LIN {X 0,Y 417.232,Z 275.449,A -85,B 0,C 180,E1 -10353.741,E2 -10353.741} C_VEL
LIN {X 0,Y 417.731,Z 261.552,A -85,B 0,C 180,E1 -10354.25,E2 -10354.25} C_VEL
LIN {X 0,Y 418.018,Z 247.194,A -85,B 0,C 180,E1 -10354.579,E2 -10354.579} C_VEL
LIN {X 0,Y 419.623,Z 143.147,A -85,B 0,C 180,E1 -10356.374,E2 -10356.374} C_VEL
LIN {X 0,Y 414.972,Z 121.368,A -85,B 0,C 180,E1 -10357.003,E2 -10357.003} C_VEL
LIN {X 0,Y 414.069,Z 118.736,A -85,B 0,C 180,E1 -10357.128,E2 -10357.128} C_VEL
LIN {X 0,Y 411.674,Z 106.755,A -85,B 0,C 180,E1 -10359.828,E2 -10359.828} C_VEL
LIN {X 0,Y 411.268,Z 104.886,A -85,B 0,C 180,E1 -10360.273,E2 -10360.273} C_VEL
LIN {X 0,Y 411.343,Z 104.878,A -85,B 0,C 180,E1 -10363.149,E2 -10363.149} C_VEL
LIN {X 0,Y 411.264,Z 104.878,A -85,B 0,C 180,E1 -10366.887,E2 -10366.887} C_VEL
LIN {X 0,Y 411.218,Z 104.885,A -85,B 0,C 180,E1 -10369.986,E2 -10369.986} C_VEL
LIN {X 0,Y 411.195,Z 104.89,A -85,B 0,C 180,E1 -10373.146,E2 -10373.146} C_VEL
LIN {X 0,Y 411.203,Z 104.885,A -85,B 0,C 180,E1 -10376.382,E2 -10376.382} C_VEL
LIN {X 0,Y 411.177,Z 104.89,A -85,B 0,C 180,E1 -10379.713,E2 -10379.713} C_VEL
LIN {X 0,Y 411.172,Z 104.896,A -85,B 0,C 180,E1 -10383.157,E2 -10383.157} C_VEL
LIN {X 0,Y 411.199,Z 104.889,A -85,B 0,C 180,E1 -10386.739,E2 -10386.739} C_VEL
LIN {X 0,Y 411.205,Z 104.885,A -85,B 0,C 180,E1 -10389.734,E2 -10389.734} C_VEL
LIN {X 0,Y 411.197,Z 104.889,A -85,B 0,C 180,E1 -10393.128,E2 -10393.128} C_VEL
LIN {X 0,Y 411.218,Z 104.883,A -85,B 0,C 180,E1 -10395.872,E2 -10395.872} C_VEL
LIN {X 0,Y 411.184,Z 104.887,A -85,B 0,C 180,E1 -10399.502,E2 -10399.502} C_VEL
LIN {X 0,Y 411.178,Z 104.89,A -85,B 0,C 180,E1 -10402.03,E2 -10402.03} C_VEL
LIN {X 0,Y 411.179,Z 104.888,A -85,B 0,C 180,E1 -10405.669,E2 -10405.669} C_VEL
LIN {X 0,Y 411.176,Z 104.888,A -85,B 0,C 180,E1 -10409.156,E2 -10409.156} C_VEL
LIN {X 0,Y 411.236,Z 104.884,A -85,B 0,C 180,E1 -10412.525,E2 -10412.525} C_VEL
LIN {X 0,Y 411.21,Z 104.887,A -85,B 0,C 180,E1 -10415.788,E2 -10415.788} C_VEL
LIN {X 0,Y 411.224,Z 104.882,A -85,B 0,C 180,E1 -10418.972,E2 -10418.972} C_VEL
LIN {X 0,Y 411.235,Z 104.886,A -85,B 0,C 180,E1 -10422.088,E2 -10422.088} C_VEL
LIN {X 0,Y 411.249,Z 104.88,A -85,B 0,C 180,E1 -10425.151,E2 -10425.151} C_VEL
LIN {X 0,Y 411.284,Z 104.877,A -85,B 0,C 180,E1 -10428.171,E2 -10428.171} C_VEL
LIN {X 0,Y 411.467,Z 104.853,A -85,B 0,C 180,E1 -10432.15,E2 -10432.15} C_VEL
LIN {X 0,Y 411.465,Z 104.854,A -85,B 0,C 180,E1 -10434.121,E2 -10434.121} C_VEL
LIN {X 0,Y 411.503,Z 104.848,A -85,B 0,C 180,E1 -10438.046,E2 -10438.046} C_VEL
LIN {X 0,Y 411.633,Z 104.832,A -85,B 0,C 180,E1 -10440.003,E2 -10440.003} C_VEL
LIN {X 0,Y 411.457,Z 104.857,A -85,B 0,C 180,E1 -10442.94,E2 -10442.94} C_VEL
LIN {X 0,Y 411.452,Z 104.858,A -85,B 0,C 180,E1 -10446.87,E2 -10446.87} C_VEL
LIN {X 0,Y 411.286,Z 104.875,A -85,B 0,C 180,E1 -10449.842,E2 -10449.842} C_VEL
LIN {X 0,Y 411.298,Z 104.878,A -85,B 0,C 180,E1 -10453.107,E2 -10453.107} C_VEL
LIN {X 0,Y 411.252,Z 104.885,A -85,B 0,C 180,E1 -10456.892,E2 -10456.892} C_VEL
LIN {X 0,Y 411.226,Z 104.883,A -85,B 0,C 180,E1 -10459.99,E2 -10459.99} C_VEL
LIN {X 0,Y 411.199,Z 104.887,A -85,B 0,C 180,E1 -10463.15,E2 -10463.15} C_VEL
LIN {X 0,Y 411.235,Z 104.886,A -85,B 0,C 180,E1 -10466.384,E2 -10466.384} C_VEL
LIN {X 0,Y 411.198,Z 104.886,A -85,B 0,C 180,E1 -10469.715,E2 -10469.715} C_VEL
LIN {X 0,Y 411.205,Z 104.885,A -85,B 0,C 180,E1 -10473.158,E2 -10473.158} C_VEL
LIN {X 0,Y 411.192,Z 104.889,A -85,B 0,C 180,E1 -10476.555,E2 -10476.555} C_VEL
LIN {X 0,Y 411.212,Z 104.887,A -85,B 0,C 180,E1 -10479.73,E2 -10479.73} C_VEL
LIN {X 0,Y 411.173,Z 104.889,A -85,B 0,C 180,E1 -10483.136,E2 -10483.136} C_VEL
LIN {X 0,Y 411.168,Z 104.896,A -85,B 0,C 180,E1 -10485.884,E2 -10485.884} C_VEL
LIN {X 0,Y 411.164,Z 104.89,A -85,B 0,C 180,E1 -10488.774,E2 -10488.774} C_VEL
LIN {X 0,Y 411.191,Z 104.89,A -85,B 0,C 180,E1 -10492.028,E2 -10492.028} C_VEL
LIN {X 0,Y 411.208,Z 104.891,A -85,B 0,C 180,E1 -10495.669,E2 -10495.669} C_VEL
LIN {X 0,Y 411.193,Z 104.891,A -85,B 0,C 180,E1 -10499.155,E2 -10499.155} C_VEL
LIN {X 0,Y 411.272,Z 104.953,A -85,B 0,C 180,E1 -10500.26,E2 -10500.26} C_VEL
LIN {X 0,Y 414.489,Z 119.861,A -85,B 0,C 180,E1 -10503.302,E2 -10503.302} C_VEL
LIN {X 0,Y 415.269,Z 124.242,A -85,B 0,C 180,E1 -10504.166,E2 -10504.166} C_VEL
LIN {X 0,Y 414.279,Z 139.428,A -85,B 0,C 180,E1 -10506.93,E2 -10506.93} C_VEL
LIN {X 0,Y 419.416,Z 170.231,A -85,B 0,C 180,E1 -10507.745,E2 -10507.745} C_VEL
LIN {X 0,Y 417.748,Z 278.062,A -85,B 0,C 180,E1 -10509.634,E2 -10509.634} C_VEL
LIN {X 0,Y 417.18,Z 292.545,A -85,B 0,C 180,E1 -10510.087,E2 -10510.087} C_VEL
LIN {X 0,Y 416.418,Z 306.482,A -85,B 0,C 180,E1 -10510.723,E2 -10510.723} C_VEL
LIN {X 0,Y 415.61,Z 319.466,A -85,B 0,C 180,E1 -10511.516,E2 -10511.516} C_VEL
LIN {X 0,Y 414.604,Z 332.073,A -85,B 0,C 180,E1 -10512.491,E2 -10512.491} C_VEL
LIN {X 0,Y 413.679,Z 343.587,A -85,B 0,C 180,E1 -10513.596,E2 -10513.596} C_VEL
LIN {X 0,Y 412.83,Z 353.163,A -85,B 0,C 180,E1 -10514.702,E2 -10514.702} C_VEL
LIN {X 0,Y 412.028,Z 363.834,A -85,B 0,C 180,E1 -10516.186,E2 -10516.186} C_VEL
LIN {X 0,Y 411.333,Z 372.623,A -85,B 0,C 180,E1 -10517.67,E2 -10517.67} C_VEL
LIN {X 0,Y 410.717,Z 381.037,A -85,B 0,C 180,E1 -10519.402,E2 -10519.402} C_VEL
LIN {X 0,Y 410.328,Z 387.778,A -85,B 0,C 180,E1 -10521.134,E2 -10521.134} C_VEL
LIN {X 0,Y 410.063,Z 393.746,A -85,B 0,C 180,E1 -10523.111,E2 -10523.111} C_VEL
LIN {X 0,Y 409.972,Z 398.111,A -85,B 0,C 180,E1 -10525.084,E2 -10525.084} C_VEL
LIN {X 0,Y 409.917,Z 401.01,A -85,B 0,C 180,E1 -10527.053,E2 -10527.053} C_VEL
LIN {X 0,Y 409.937,Z 402.528,A -85,B 0,C 180,E1 -10529.019,E2 -10529.019} C_VEL
LIN {X 0,Y 409.937,Z 402.7,A -85,B 0,C 180,E1 -10530.984,E2 -10530.984} C_VEL
LIN {X 0,Y 409.913,Z 401.537,A -85,B 0,C 180,E1 -10532.95,E2 -10532.95} C_VEL
LIN {X 0,Y 409.982,Z 399.026,A -85,B 0,C 180,E1 -10534.918,E2 -10534.918} C_VEL
LIN {X 0,Y 410.092,Z 395.089,A -85,B 0,C 180,E1 -10536.891,E2 -10536.891} C_VEL
LIN {X 0,Y 410.402,Z 389.593,A -85,B 0,C 180,E1 -10538.867,E2 -10538.867} C_VEL
LIN {X 0,Y 410.803,Z 383.407,A -85,B 0,C 180,E1 -10540.599,E2 -10540.599} C_VEL
LIN {X 0,Y 411.606,Z 375.714,A -85,B 0,C 180,E1 -10542.325,E2 -10542.325} C_VEL
LIN {X 0,Y 412.283,Z 367.712,A -85,B 0,C 180,E1 -10543.808,E2 -10543.808} C_VEL
LIN {X 0,Y 413.236,Z 358.091,A -85,B 0,C 180,E1 -10545.286,E2 -10545.286} C_VEL
LIN {X 0,Y 414.334,Z 347.445,A -85,B 0,C 180,E1 -10546.634,E2 -10546.634} C_VEL
LIN {X 0,Y 415.594,Z 335.694,A -85,B 0,C 180,E1 -10547.85,E2 -10547.85} C_VEL
LIN {X 0,Y 416.616,Z 324.265,A -85,B 0,C 180,E1 -10548.819,E2 -10548.819} C_VEL
LIN {X 0,Y 417.625,Z 311.778,A -85,B 0,C 180,E1 -10549.669,E2 -10549.669} C_VEL
LIN {X 0,Y 418.607,Z 298.001,A -85,B 0,C 180,E1 -10550.389,E2 -10550.389} C_VEL
LIN {X 0,Y 419.4,Z 284.502,A -85,B 0,C 180,E1 -10550.894,E2 -10550.894} C_VEL
LIN {X 0,Y 419.898,Z 271.046,A -85,B 0,C 180,E1 -10551.221,E2 -10551.221} C_VEL
LIN {X 0,Y 421.535,Z 169.575,A -85,B 0,C 180,E1 -10553.015,E2 -10553.015} C_VEL
LIN {X 0,Y 417.055,Z 146.34,A -85,B 0,C 180,E1 -10553.757,E2 -10553.757} C_VEL
LIN {X 0,Y 415.437,Z 138.972,A -85,B 0,C 180,E1 -10554.021,E2 -10554.021} C_VEL
LIN {X 0,Y 416.422,Z 128.312,A -85,B 0,C 180,E1 -10556.029,E2 -10556.029} C_VEL
LIN {X 0,Y 414.54,Z 118.327,A -85,B 0,C 180,E1 -10558.162,E2 -10558.162} C_VEL
LIN {X 0,Y 411.687,Z 106.654,A -85,B 0,C 180,E1 -10560.808,E2 -10560.808} C_VEL
LIN {X 0,Y 411.202,Z 104.895,A -85,B 0,C 180,E1 -10561.238,E2 -10561.238} C_VEL
LIN {X 0,Y 411.205,Z 104.889,A -85,B 0,C 180,E1 -10564.335,E2 -10564.335} C_VEL
LIN {X 0,Y 411.202,Z 104.887,A -85,B 0,C 180,E1 -10566.742,E2 -10566.742} C_VEL
LIN {X 0,Y 411.209,Z 104.886,A -85,B 0,C 180,E1 -10569.724,E2 -10569.724} C_VEL
LIN {X 0,Y 411.185,Z 104.889,A -85,B 0,C 180,E1 -10573.134,E2 -10573.134} C_VEL
LIN {X 0,Y 411.182,Z 104.893,A -85,B 0,C 180,E1 -10575.881,E2 -10575.881} C_VEL
LIN {X 0,Y 411.174,Z 104.875,A -85,B 0,C 180,E1 -10578.772,E2 -10578.772} C_VEL
LIN {X 0,Y 411.2,Z 104.886,A -85,B 0,C 180,E1 -10582.024,E2 -10582.024} C_VEL
LIN {X 0,Y 411.217,Z 104.887,A -85,B 0,C 180,E1 -10585.122,E2 -10585.122} C_VEL
LIN {X 0,Y 411.179,Z 104.888,A -85,B 0,C 180,E1 -10588.001,E2 -10588.001} C_VEL
LIN {X 0,Y 411.207,Z 104.886,A -85,B 0,C 180,E1 -10591.407,E2 -10591.407} C_VEL
LIN {X 0,Y 411.241,Z 104.885,A -85,B 0,C 180,E1 -10594.928,E2 -10594.928} C_VEL
LIN {X 0,Y 411.218,Z 104.885,A -85,B 0,C 180,E1 -10597.912,E2 -10597.912} C_VEL
LIN {X 0,Y 411.232,Z 104.885,A -85,B 0,C 180,E1 -10601.049,E2 -10601.049} C_VEL
LIN {X 0,Y 411.266,Z 104.873,A -85,B 0,C 180,E1 -10604.129,E2 -10604.129} C_VEL
LIN {X 0,Y 411.315,Z 104.87,A -85,B 0,C 180,E1 -10607.163,E2 -10607.163} C_VEL
LIN {X 0,Y 411.301,Z 104.876,A -85,B 0,C 180,E1 -10610.159,E2 -10610.159} C_VEL
LIN {X 0,Y 411.402,Z 104.859,A -85,B 0,C 180,E1 -10613.129,E2 -10613.129} C_VEL
LIN {X 0,Y 411.308,Z 104.873,A -85,B 0,C 180,E1 -10615.096,E2 -10615.096} C_VEL
LIN {X 0,Y 411.516,Z 104.846,A -85,B 0,C 180,E1 -10618.039,E2 -10618.039} C_VEL
LIN {X 0,Y 411.643,Z 104.834,A -85,B 0,C 180,E1 -10619.997,E2 -10619.997} C_VEL
LIN {X 0,Y 411.456,Z 104.855,A -85,B 0,C 180,E1 -10622.934,E2 -10622.934} C_VEL
LIN {X 0,Y 411.428,Z 104.858,A -85,B 0,C 180,E1 -10626.864,E2 -10626.864} C_VEL
LIN {X 0,Y 411.294,Z 104.874,A -85,B 0,C 180,E1 -10629.835,E2 -10629.835} C_VEL
LIN {X 0,Y 411.307,Z 104.872,A -85,B 0,C 180,E1 -10633.1,E2 -10633.1} C_VEL
LIN {X 0,Y 411.257,Z 104.877,A -85,B 0,C 180,E1 -10636.885,E2 -10636.885} C_VEL
LIN {X 0,Y 411.228,Z 104.88,A -85,B 0,C 180,E1 -10639.983,E2 -10639.983} C_VEL
LIN {X 0,Y 411.191,Z 104.889,A -85,B 0,C 180,E1 -10643.144,E2 -10643.144} C_VEL
LIN {X 0,Y 411.227,Z 104.881,A -85,B 0,C 180,E1 -10646.377,E2 -10646.377} C_VEL
LIN {X 0,Y 411.192,Z 104.875,A -85,B 0,C 180,E1 -10649.709,E2 -10649.709} C_VEL
LIN {X 0,Y 411.196,Z 104.884,A -85,B 0,C 180,E1 -10653.152,E2 -10653.152} C_VEL
LIN {X 0,Y 411.179,Z 104.895,A -85,B 0,C 180,E1 -10656.548,E2 -10656.548} C_VEL
LIN {X 0,Y 411.194,Z 104.891,A -85,B 0,C 180,E1 -10659.723,E2 -10659.723} C_VEL
LIN {X 0,Y 411.156,Z 104.897,A -85,B 0,C 180,E1 -10663.13,E2 -10663.13} C_VEL
LIN {X 0,Y 411.16,Z 104.933,A -85,B 0,C 180,E1 -10666.378,E2 -10666.378} C_VEL
LIN {X 0,Y 413.745,Z 115.767,A -85,B 0,C 180,E1 -10669.096,E2 -10669.096} C_VEL
LIN {X 0,Y 414.472,Z 119.37,A -85,B 0,C 180,E1 -10669.967,E2 -10669.967} C_VEL
LIN {X 0,Y 418.585,Z 129.465,A -85,B 0,C 180,E1 -10670.453,E2 -10670.453} C_VEL
LIN {X 0,Y 422,Z 144.277,A -85,B 0,C 180,E1 -10670.966,E2 -10670.966} C_VEL
LIN {X 0,Y 419.998,Z 256.023,A -85,B 0,C 180,E1 -10672.956,E2 -10672.956} C_VEL
LIN {X 0,Y 419.376,Z 270.729,A -85,B 0,C 180,E1 -10673.419,E2 -10673.419} C_VEL
LIN {X 0,Y 418.604,Z 285.001,A -85,B 0,C 180,E1 -10674.085,E2 -10674.085} C_VEL
LIN {X 0,Y 417.765,Z 296.896,A -85,B 0,C 180,E1 -10674.816,E2 -10674.816} C_VEL
LIN {X 0,Y 416.802,Z 308.452,A -85,B 0,C 180,E1 -10675.704,E2 -10675.704} C_VEL
LIN {X 0,Y 415.673,Z 320.161,A -85,B 0,C 180,E1 -10676.811,E2 -10676.811} C_VEL
LIN {X 0,Y 414.582,Z 330.837,A -85,B 0,C 180,E1 -10678.042,E2 -10678.042} C_VEL
LIN {X 0,Y 413.566,Z 340.245,A -85,B 0,C 180,E1 -10679.347,E2 -10679.347} C_VEL
LIN {X 0,Y 412.538,Z 349.792,A -85,B 0,C 180,E1 -10680.952,E2 -10680.952} C_VEL
LIN {X 0,Y 411.715,Z 357.654,A -85,B 0,C 180,E1 -10682.568,E2 -10682.568} C_VEL
LIN {X 0,Y 411.116,Z 363.963,A -85,B 0,C 180,E1 -10684.155,E2 -10684.155} C_VEL
LIN {X 0,Y 410.655,Z 369.11,A -85,B 0,C 180,E1 -10685.747,E2 -10685.747} C_VEL
LIN {X 0,Y 410.33,Z 373.842,A -85,B 0,C 180,E1 -10687.639,E2 -10687.639} C_VEL
LIN {X 0,Y 410.094,Z 376.27,A -85,B 0,C 180,E1 -10688.905,E2 -10688.905} C_VEL
LIN {X 0,Y 409.88,Z 378.977,A -85,B 0,C 180,E1 -10690.986,E2 -10690.986} C_VEL
LIN {X 0,Y 409.79,Z 380.163,A -85,B 0,C 180,E1 -10693.048,E2 -10693.048} C_VEL
LIN {X 0,Y 409.814,Z 380.219,A -85,B 0,C 180,E1 -10694.073,E2 -10694.073} C_VEL
LIN {X 0,Y 409.789,Z 379.28,A -85,B 0,C 180,E1 -10696.106,E2 -10696.106} C_VEL
LIN {X 0,Y 409.959,Z 376.935,A -85,B 0,C 180,E1 -10698.127,E2 -10698.127} C_VEL
LIN {X 0,Y 410.151,Z 373.162,A -85,B 0,C 180,E1 -10700.132,E2 -10700.132} C_VEL
LIN {X 0,Y 410.382,Z 369.027,A -85,B 0,C 180,E1 -10701.722,E2 -10701.722} C_VEL
LIN {X 0,Y 409.855,Z 366.761,A -85,B 0,C 180,E1 -10702.481,E2 -10702.481} C_VEL
LIN {X 0,Y 407.293,Z 362.771,A -85,B 0,C 180,E1 -10703.703,E2 -10703.703} C_VEL
LIN {X 0,Y 404.787,Z 358.223,A -85,B 0,C 180,E1 -10704.898,E2 -10704.898} C_VEL
LIN {X 0,Y 404.353,Z 355.068,A -85,B 0,C 180,E1 -10705.605,E2 -10705.605} C_VEL
LIN {X 0,Y 405.15,Z 346.404,A -85,B 0,C 180,E1 -10707.264,E2 -10707.264} C_VEL
LIN {X 0,Y 406.01,Z 336.893,A -85,B 0,C 180,E1 -10708.759,E2 -10708.759} C_VEL
LIN {X 0,Y 406.95,Z 326.374,A -85,B 0,C 180,E1 -10710.122,E2 -10710.122} C_VEL
LIN {X 0,Y 407.826,Z 315.863,A -85,B 0,C 180,E1 -10711.251,E2 -10711.251} C_VEL
LIN {X 0,Y 408.785,Z 303.467,A -85,B 0,C 180,E1 -10712.339,E2 -10712.339} C_VEL
LIN {X 0,Y 409.661,Z 291.236,A -85,B 0,C 180,E1 -10713.195,E2 -10713.195} C_VEL
LIN {X 0,Y 410.372,Z 277.79,A -85,B 0,C 180,E1 -10713.927,E2 -10713.927} C_VEL
LIN {X 0,Y 410.892,Z 263.957,A -85,B 0,C 180,E1 -10714.474,E2 -10714.474} C_VEL
LIN {X 0,Y 411.246,Z 249.63,A -85,B 0,C 180,E1 -10714.839,E2 -10714.839} C_VEL
LIN {X 0,Y 412.995,Z 144.462,A -85,B 0,C 180,E1 -10716.679,E2 -10716.679} C_VEL
LIN {X 0,Y 408.494,Z 123.578,A -85,B 0,C 180,E1 -10717.293,E2 -10717.293} C_VEL
LIN {X 0,Y 406.945,Z 119.084,A -85,B 0,C 180,E1 -10717.459,E2 -10717.459} C_VEL
LIN {X 0,Y 404.703,Z 108.046,A -85,B 0,C 180,E1 -10719.999,E2 -10719.999} C_VEL
LIN {X 0,Y 404.227,Z 105.761,A -85,B 0,C 180,E1 -10720.58,E2 -10720.58} C_VEL
LIN {X 0,Y 404.284,Z 105.757,A -85,B 0,C 180,E1 -10723.244,E2 -10723.244} C_VEL
LIN {X 0,Y 404.211,Z 105.758,A -85,B 0,C 180,E1 -10727.191,E2 -10727.191} C_VEL
LIN {X 0,Y 404.17,Z 105.761,A -85,B 0,C 180,E1 -10730.35,E2 -10730.35} C_VEL
LIN {X 0,Y 404.149,Z 105.769,A -85,B 0,C 180,E1 -10733.574,E2 -10733.574} C_VEL
LIN {X 0,Y 404.16,Z 105.765,A -85,B 0,C 180,E1 -10736.878,E2 -10736.878} C_VEL
LIN {X 0,Y 404.121,Z 105.767,A -85,B 0,C 180,E1 -10740.285,E2 -10740.285} C_VEL
LIN {X 0,Y 404.112,Z 105.769,A -85,B 0,C 180,E1 -10743.813,E2 -10743.813} C_VEL
LIN {X 0,Y 404.145,Z 105.77,A -85,B 0,C 180,E1 -10746.885,E2 -10746.885} C_VEL
LIN {X 0,Y 404.165,Z 105.762,A -85,B 0,C 180,E1 -10750.09,E2 -10750.09} C_VEL
LIN {X 0,Y 404.171,Z 105.765,A -85,B 0,C 180,E1 -10753.093,E2 -10753.093} C_VEL
LIN {X 0,Y 404.19,Z 105.759,A -85,B 0,C 180,E1 -10755.938,E2 -10755.938} C_VEL
LIN {X 0,Y 404.137,Z 105.772,A -85,B 0,C 180,E1 -10758.643,E2 -10758.643} C_VEL
LIN {X 0,Y 404.135,Z 105.765,A -85,B 0,C 180,E1 -10761.493,E2 -10761.493} C_VEL
LIN {X 0,Y 404.158,Z 105.764,A -85,B 0,C 180,E1 -10764.987,E2 -10764.987} C_VEL
LIN {X 0,Y 404.125,Z 105.771,A -85,B 0,C 180,E1 -10768.557,E2 -10768.557} C_VEL
LIN {X 0,Y 404.174,Z 105.765,A -85,B 0,C 180,E1 -10772.004,E2 -10772.004} C_VEL
LIN {X 0,Y 404.158,Z 105.763,A -85,B 0,C 180,E1 -10775.338,E2 -10775.338} C_VEL
LIN {X 0,Y 404.182,Z 105.761,A -85,B 0,C 180,E1 -10778.587,E2 -10778.587} C_VEL
LIN {X 0,Y 404.197,Z 105.763,A -85,B 0,C 180,E1 -10781.765,E2 -10781.765} C_VEL
LIN {X 0,Y 404.195,Z 105.758,A -85,B 0,C 180,E1 -10784.886,E2 -10784.886} C_VEL
LIN {X 0,Y 404.254,Z 105.755,A -85,B 0,C 180,E1 -10787.962,E2 -10787.962} C_VEL
LIN {X 0,Y 404.419,Z 105.732,A -85,B 0,C 180,E1 -10792.103,E2 -10792.103} C_VEL
LIN {X 0,Y 404.413,Z 105.733,A -85,B 0,C 180,E1 -10794.018,E2 -10794.018} C_VEL
LIN {X 0,Y 404.472,Z 105.725,A -85,B 0,C 180,E1 -10798.012,E2 -10798.012} C_VEL
LIN {X 0,Y 404.602,Z 105.708,A -85,B 0,C 180,E1 -10800.003,E2 -10800.003} C_VEL
LIN {X 0,Y 404.414,Z 105.734,A -85,B 0,C 180,E1 -10802.992,E2 -10802.992} C_VEL
LIN {X 0,Y 404.403,Z 105.737,A -85,B 0,C 180,E1 -10806.99,E2 -10806.99} C_VEL
LIN {X 0,Y 404.251,Z 105.751,A -85,B 0,C 180,E1 -10810.015,E2 -10810.015} C_VEL
LIN {X 0,Y 404.26,Z 105.754,A -85,B 0,C 180,E1 -10813.214,E2 -10813.214} C_VEL
LIN {X 0,Y 404.21,Z 105.761,A -85,B 0,C 180,E1 -10817.01,E2 -10817.01} C_VEL
LIN {X 0,Y 404.159,Z 105.765,A -85,B 0,C 180,E1 -10820.355,E2 -10820.355} C_VEL
LIN {X 0,Y 404.166,Z 105.762,A -85,B 0,C 180,E1 -10823.577,E2 -10823.577} C_VEL
LIN {X 0,Y 404.181,Z 105.76,A -85,B 0,C 180,E1 -10825.769,E2 -10825.769} C_VEL
LIN {X 0,Y 404.193,Z 105.76,A -85,B 0,C 180,E1 -10828.002,E2 -10828.002} C_VEL
LIN {X 0,Y 404.137,Z 105.765,A -85,B 0,C 180,E1 -10831.561,E2 -10831.561} C_VEL
LIN {X 0,Y 404.184,Z 105.76,A -85,B 0,C 180,E1 -10835.019,E2 -10835.019} C_VEL
LIN {X 0,Y 404.153,Z 105.764,A -85,B 0,C 180,E1 -10838.76,E2 -10838.76} C_VEL
LIN {X 0,Y 404.122,Z 105.769,A -85,B 0,C 180,E1 -10841.602,E2 -10841.602} C_VEL
LIN {X 0,Y 404.146,Z 105.765,A -85,B 0,C 180,E1 -10844.524,E2 -10844.524} C_VEL
LIN {X 0,Y 404.137,Z 105.766,A -85,B 0,C 180,E1 -10847.298,E2 -10847.298} C_VEL
LIN {X 0,Y 404.171,Z 105.766,A -85,B 0,C 180,E1 -10849.958,E2 -10849.958} C_VEL
LIN {X 0,Y 404.137,Z 105.766,A -85,B 0,C 180,E1 -10853.128,E2 -10853.128} C_VEL
LIN {X 0,Y 404.148,Z 105.769,A -85,B 0,C 180,E1 -10856.19,E2 -10856.19} C_VEL
LIN {X 0,Y 404.216,Z 105.941,A -85,B 0,C 180,E1 -10859.994,E2 -10859.994} C_VEL
LIN {X 0,Y 407.453,Z 120.771,A -85,B 0,C 180,E1 -10863.08,E2 -10863.08} C_VEL
LIN {X 0,Y 408.357,Z 126.76,A -85,B 0,C 180,E1 -10864.273,E2 -10864.273} C_VEL
LIN {X 0,Y 407.418,Z 139.188,A -85,B 0,C 180,E1 -10866.567,E2 -10866.567} C_VEL
LIN {X 0,Y 412.694,Z 170.64,A -85,B 0,C 180,E1 -10867.427,E2 -10867.427} C_VEL
LIN {X 0,Y 411.015,Z 277.225,A -85,B 0,C 180,E1 -10869.318,E2 -10869.318} C_VEL
LIN {X 0,Y 410.441,Z 291.926,A -85,B 0,C 180,E1 -10869.779,E2 -10869.779} C_VEL
LIN {X 0,Y 409.66,Z 305.399,A -85,B 0,C 180,E1 -10870.393,E2 -10870.393} C_VEL
LIN {X 0,Y 408.764,Z 318.886,A -85,B 0,C 180,E1 -10871.218,E2 -10871.218} C_VEL
LIN {X 0,Y 407.786,Z 331.318,A -85,B 0,C 180,E1 -10872.189,E2 -10872.189} C_VEL
LIN {X 0,Y 406.78,Z 342.927,A -85,B 0,C 180,E1 -10873.309,E2 -10873.309} C_VEL
LIN {X 0,Y 405.899,Z 352.583,A -85,B 0,C 180,E1 -10874.434,E2 -10874.434} C_VEL
LIN {X 0,Y 405.053,Z 363.318,A -85,B 0,C 180,E1 -10875.943,E2 -10875.943} C_VEL
LIN {X 0,Y 404.36,Z 372.163,A -85,B 0,C 180,E1 -10877.454,E2 -10877.454} C_VEL
LIN {X 0,Y 403.677,Z 380.63,A -85,B 0,C 180,E1 -10879.215,E2 -10879.215} C_VEL
LIN {X 0,Y 403.277,Z 387.426,A -85,B 0,C 180,E1 -10880.978,E2 -10880.978} C_VEL
LIN {X 0,Y 403.041,Z 392.086,A -85,B 0,C 180,E1 -10882.487,E2 -10882.487} C_VEL
LIN {X 0,Y 402.858,Z 396.38,A -85,B 0,C 180,E1 -10884.252,E2 -10884.252} C_VEL
LIN {X 0,Y 402.827,Z 399.477,A -85,B 0,C 180,E1 -10886,E2 -10886} C_VEL
LIN {X 0,Y 402.864,Z 401.709,A -85,B 0,C 180,E1 -10888.002,E2 -10888.002} C_VEL
LIN {X 0,Y 402.855,Z 402.579,A -85,B 0,C 180,E1 -10890.001,E2 -10890.001} C_VEL
LIN {X 0,Y 402.864,Z 402.111,A -85,B 0,C 180,E1 -10892.001,E2 -10892.001} C_VEL
LIN {X 0,Y 402.828,Z 400.306,A -85,B 0,C 180,E1 -10894.003,E2 -10894.003} C_VEL
LIN {X 0,Y 402.927,Z 397.133,A -85,B 0,C 180,E1 -10896.009,E2 -10896.009} C_VEL
LIN {X 0,Y 403.158,Z 392.478,A -85,B 0,C 180,E1 -10898.018,E2 -10898.018} C_VEL
LIN {X 0,Y 403.607,Z 386.192,A -85,B 0,C 180,E1 -10900.029,E2 -10900.029} C_VEL
LIN {X 0,Y 404.266,Z 379.215,A -85,B 0,C 180,E1 -10901.788,E2 -10901.788} C_VEL
LIN {X 0,Y 405.032,Z 370.917,A -85,B 0,C 180,E1 -10903.487,E2 -10903.487} C_VEL
LIN {X 0,Y 405.998,Z 361.607,A -85,B 0,C 180,E1 -10905.051,E2 -10905.051} C_VEL
LIN {X 0,Y 407.193,Z 350.766,A -85,B 0,C 180,E1 -10906.547,E2 -10906.547} C_VEL
LIN {X 0,Y 408.421,Z 339.795,A -85,B 0,C 180,E1 -10907.786,E2 -10907.786} C_VEL
LIN {X 0,Y 409.635,Z 327.789,A -85,B 0,C 180,E1 -10908.896,E2 -10908.896} C_VEL
LIN {X 0,Y 410.805,Z 314.957,A -85,B 0,C 180,E1 -10909.842,E2 -10909.842} C_VEL
LIN {X 0,Y 411.858,Z 301.474,A -85,B 0,C 180,E1 -10910.608,E2 -10910.608} C_VEL
LIN {X 0,Y 412.702,Z 287.662,A -85,B 0,C 180,E1 -10911.184,E2 -10911.184} C_VEL
LIN {X 0,Y 413.377,Z 273.369,A -85,B 0,C 180,E1 -10911.572,E2 -10911.572} C_VEL
LIN {X 0,Y 415.22,Z 170.983,A -85,B 0,C 180,E1 -10913.412,E2 -10913.412} C_VEL
LIN {X 0,Y 410.929,Z 148.637,A -85,B 0,C 180,E1 -10914.145,E2 -10914.145} C_VEL
LIN {X 0,Y 408.768,Z 138.757,A -85,B 0,C 180,E1 -10914.506,E2 -10914.506} C_VEL
LIN {X 0,Y 409.619,Z 129.836,A -85,B 0,C 180,E1 -10916.22,E2 -10916.22} C_VEL
LIN {X 0,Y 407.649,Z 119.651,A -85,B 0,C 180,E1 -10918.444,E2 -10918.444} C_VEL
LIN {X 0,Y 404.757,Z 108.233,A -85,B 0,C 180,E1 -10921.103,E2 -10921.103} C_VEL
LIN {X 0,Y 404.15,Z 105.772,A -85,B 0,C 180,E1 -10921.716,E2 -10921.716} C_VEL
LIN {X 0,Y 404.187,Z 105.762,A -85,B 0,C 180,E1 -10925.017,E2 -10925.017} C_VEL
LIN {X 0,Y 404.156,Z 105.768,A -85,B 0,C 180,E1 -10928.758,E2 -10928.758} C_VEL
LIN {X 0,Y 404.131,Z 105.767,A -85,B 0,C 180,E1 -10931.598,E2 -10931.598} C_VEL
LIN {X 0,Y 404.159,Z 105.766,A -85,B 0,C 180,E1 -10934.521,E2 -10934.521} C_VEL
LIN {X 0,Y 404.149,Z 105.766,A -85,B 0,C 180,E1 -10937.295,E2 -10937.295} C_VEL
LIN {X 0,Y 404.147,Z 105.76,A -85,B 0,C 180,E1 -10939.95,E2 -10939.95} C_VEL
LIN {X 0,Y 404.148,Z 105.763,A -85,B 0,C 180,E1 -10943.125,E2 -10943.125} C_VEL
LIN {X 0,Y 404.152,Z 105.764,A -85,B 0,C 180,E1 -10946.186,E2 -10946.186} C_VEL
LIN {X 0,Y 404.158,Z 105.767,A -85,B 0,C 180,E1 -10949.713,E2 -10949.713} C_VEL
LIN {X 0,Y 404.149,Z 105.765,A -85,B 0,C 180,E1 -10953.117,E2 -10953.117} C_VEL
LIN {X 0,Y 404.174,Z 105.756,A -85,B 0,C 180,E1 -10956.423,E2 -10956.423} C_VEL
LIN {X 0,Y 404.205,Z 105.751,A -85,B 0,C 180,E1 -10959.872,E2 -10959.872} C_VEL
LIN {X 0,Y 404.229,Z 105.754,A -85,B 0,C 180,E1 -10962.991,E2 -10962.991} C_VEL
LIN {X 0,Y 404.295,Z 105.747,A -85,B 0,C 180,E1 -10966.936,E2 -10966.936} C_VEL
LIN {X 0,Y 404.267,Z 105.751,A -85,B 0,C 180,E1 -10969.986,E2 -10969.986} C_VEL
LIN {X 0,Y 404.353,Z 105.738,A -85,B 0,C 180,E1 -10973.009,E2 -10973.009} C_VEL
LIN {X 0,Y 404.279,Z 105.749,A -85,B 0,C 180,E1 -10975.01,E2 -10975.01} C_VEL
LIN {X 0,Y 404.485,Z 105.722,A -85,B 0,C 180,E1 -10978.005,E2 -10978.005} C_VEL
LIN {X 0,Y 404.613,Z 105.709,A -85,B 0,C 180,E1 -10979.997,E2 -10979.997} C_VEL
LIN {X 0,Y 404.414,Z 105.732,A -85,B 0,C 180,E1 -10982.985,E2 -10982.985} C_VEL
LIN {X 0,Y 404.374,Z 105.737,A -85,B 0,C 180,E1 -10986.984,E2 -10986.984} C_VEL
LIN {X 0,Y 404.26,Z 105.751,A -85,B 0,C 180,E1 -10990.008,E2 -10990.008} C_VEL
LIN {X 0,Y 404.268,Z 105.748,A -85,B 0,C 180,E1 -10993.207,E2 -10993.207} C_VEL
LIN {X 0,Y 404.216,Z 105.754,A -85,B 0,C 180,E1 -10997.003,E2 -10997.003} C_VEL
LIN {X 0,Y 404.161,Z 105.76,A -85,B 0,C 180,E1 -11000.347,E2 -11000.347} C_VEL
LIN {X 0,Y 404.155,Z 105.766,A -85,B 0,C 180,E1 -11003.571,E2 -11003.571} C_VEL
LIN {X 0,Y 404.175,Z 105.759,A -85,B 0,C 180,E1 -11005.762,E2 -11005.762} C_VEL
LIN {X 0,Y 404.188,Z 105.76,A -85,B 0,C 180,E1 -11007.995,E2 -11007.995} C_VEL
LIN {X 0,Y 404.13,Z 105.77,A -85,B 0,C 180,E1 -11011.554,E2 -11011.554} C_VEL
LIN {X 0,Y 404.171,Z 105.759,A -85,B 0,C 180,E1 -11015.012,E2 -11015.012} C_VEL
LIN {X 0,Y 404.136,Z 105.767,A -85,B 0,C 180,E1 -11018.753,E2 -11018.753} C_VEL
LIN {X 0,Y 404.106,Z 105.771,A -85,B 0,C 180,E1 -11021.595,E2 -11021.595} C_VEL
LIN {X 0,Y 404.127,Z 105.775,A -85,B 0,C 180,E1 -11024.518,E2 -11024.518} C_VEL
LIN {X 0,Y 404.145,Z 105.938,A -85,B 0,C 180,E1 -11025.966,E2 -11025.966} C_VEL
LIN {X 0,Y 406.975,Z 117.731,A -85,B 0,C 180,E1 -11028.986,E2 -11028.986} C_VEL
LIN {X 0,Y 407.353,Z 119.607,A -85,B 0,C 180,E1 -11029.447,E2 -11029.447} C_VEL
LIN {X 0,Y 412.681,Z 132.468,A -85,B 0,C 180,E1 -11030.092,E2 -11030.092} C_VEL
LIN {X 0,Y 415.605,Z 145.213,A -85,B 0,C 180,E1 -11030.547,E2 -11030.547} C_VEL
LIN {X 0,Y 413.545,Z 256.542,A -85,B 0,C 180,E1 -11032.565,E2 -11032.565} C_VEL
LIN {X 0,Y 412.881,Z 271.072,A -85,B 0,C 180,E1 -11033.03,E2 -11033.03} C_VEL
LIN {X 0,Y 412.037,Z 285.662,A -85,B 0,C 180,E1 -11033.724,E2 -11033.724} C_VEL
LIN {X 0,Y 410.996,Z 299.19,A -85,B 0,C 180,E1 -11034.587,E2 -11034.587} C_VEL
LIN {X 0,Y 409.814,Z 312.493,A -85,B 0,C 180,E1 -11035.681,E2 -11035.681} C_VEL
LIN {X 0,Y 408.558,Z 324.253,A -85,B 0,C 180,E1 -11036.891,E2 -11036.891} C_VEL
LIN {X 0,Y 407.368,Z 335.027,A -85,B 0,C 180,E1 -11038.25,E2 -11038.25} C_VEL
LIN {X 0,Y 406.395,Z 343.983,A -85,B 0,C 180,E1 -11039.612,E2 -11039.612} C_VEL
LIN {X 0,Y 405.331,Z 352.854,A -85,B 0,C 180,E1 -11041.238,E2 -11041.238} C_VEL
LIN {X 0,Y 404.628,Z 359.542,A -85,B 0,C 180,E1 -11042.718,E2 -11042.718} C_VEL
LIN {X 0,Y 404.024,Z 365.185,A -85,B 0,C 180,E1 -11044.221,E2 -11044.221} C_VEL
LIN {X 0,Y 403.564,Z 370.112,A -85,B 0,C 180,E1 -11045.841,E2 -11045.841} C_VEL
LIN {X 0,Y 403.269,Z 373.989,A -85,B 0,C 180,E1 -11047.454,E2 -11047.454} C_VEL
LIN {X 0,Y 402.917,Z 377.674,A -85,B 0,C 180,E1 -11049.581,E2 -11049.581} C_VEL
LIN {X 0,Y 402.851,Z 378.928,A -85,B 0,C 180,E1 -11050.641,E2 -11050.641} C_VEL
LIN {X 0,Y 402.684,Z 380.318,A -85,B 0,C 180,E1 -11052.739,E2 -11052.739} C_VEL
LIN {X 0,Y 402.697,Z 380.237,A -85,B 0,C 180,E1 -11054.823,E2 -11054.823} C_VEL
LIN {X 0,Y 402.718,Z 378.75,A -85,B 0,C 180,E1 -11056.886,E2 -11056.886} C_VEL
LIN {X 0,Y 402.95,Z 375.846,A -85,B 0,C 180,E1 -11058.938,E2 -11058.938} C_VEL
LIN {X 0,Y 403.179,Z 371.486,A -85,B 0,C 180,E1 -11060.973,E2 -11060.973} C_VEL
LIN {X 0,Y 403.609,Z 365.538,A -85,B 0,C 180,E1 -11062.997,E2 -11062.997} C_VEL
LIN {X 0,Y 404.049,Z 358.858,A -85,B 0,C 180,E1 -11064.759,E2 -11064.759} C_VEL
LIN {X 0,Y 404.353,Z 355.068,A -85,B 0,C 180,E1 -11065.605,E2 -11065.605} C_VEL
LIN {X 0,Y 403.952,Z 351.786,A -85,B 0,C 180,E1 -11066.296,E2 -11066.296} C_VEL
LIN {X 0,Y 401.644,Z 346.163,A -85,B 0,C 180,E1 -11067.415,E2 -11067.415} C_VEL
LIN {X 0,Y 399.424,Z 340.131,A -85,B 0,C 180,E1 -11068.494,E2 -11068.494} C_VEL
LIN {X 0,Y 399.159,Z 336.081,A -85,B 0,C 180,E1 -11069.112,E2 -11069.112} C_VEL
LIN {X 0,Y 400.153,Z 325.322,A -85,B 0,C 180,E1 -11070.502,E2 -11070.502} C_VEL
LIN {X 0,Y 401.147,Z 313.273,A -85,B 0,C 180,E1 -11071.774,E2 -11071.774} C_VEL
LIN {X 0,Y 402.14,Z 301.773,A -85,B 0,C 180,E1 -11072.753,E2 -11072.753} C_VEL
LIN {X 0,Y 403.033,Z 288.089,A -85,B 0,C 180,E1 -11073.685,E2 -11073.685} C_VEL
LIN {X 0,Y 403.723,Z 274.101,A -85,B 0,C 180,E1 -11074.398,E2 -11074.398} C_VEL
LIN {X 0,Y 404.246,Z 260.338,A -85,B 0,C 180,E1 -11074.892,E2 -11074.892} C_VEL
LIN {X 0,Y 404.624,Z 243.267,A -85,B 0,C 180,E1 -11075.262,E2 -11075.262} C_VEL
LIN {X 0,Y 406.239,Z 145.253,A -85,B 0,C 180,E1 -11077.006,E2 -11077.006} C_VEL
LIN {X 0,Y 402.23,Z 126.279,A -85,B 0,C 180,E1 -11077.572,E2 -11077.572} C_VEL
LIN {X 0,Y 399.782,Z 119.188,A -85,B 0,C 180,E1 -11077.861,E2 -11077.861} C_VEL
LIN {X 0,Y 397.204,Z 106.636,A -85,B 0,C 180,E1 -11080.834,E2 -11080.834} C_VEL
LIN {X 0,Y 397.234,Z 106.634,A -85,B 0,C 180,E1 -11083.348,E2 -11083.348} C_VEL
LIN {X 0,Y 397.19,Z 106.633,A -85,B 0,C 180,E1 -11087.176,E2 -11087.176} C_VEL
LIN {X 0,Y 397.121,Z 106.639,A -85,B 0,C 180,E1 -11090.727,E2 -11090.727} C_VEL
LIN {X 0,Y 397.105,Z 106.642,A -85,B 0,C 180,E1 -11094.018,E2 -11094.018} C_VEL
LIN {X 0,Y 397.159,Z 106.64,A -85,B 0,C 180,E1 -11097.391,E2 -11097.391} C_VEL
LIN {X 0,Y 397.054,Z 106.651,A -85,B 0,C 180,E1 -11100.883,E2 -11100.883} C_VEL
LIN {X 0,Y 397.095,Z 106.644,A -85,B 0,C 180,E1 -11104.494,E2 -11104.494} C_VEL
LIN {X 0,Y 397.118,Z 106.64,A -85,B 0,C 180,E1 -11108.271,E2 -11108.271} C_VEL
LIN {X 0,Y 397.125,Z 106.639,A -85,B 0,C 180,E1 -11111.996,E2 -11111.996} C_VEL
LIN {X 0,Y 397.147,Z 106.639,A -85,B 0,C 180,E1 -11115.058,E2 -11115.058} C_VEL
LIN {X 0,Y 397.128,Z 106.639,A -85,B 0,C 180,E1 -11118.009,E2 -11118.009} C_VEL
LIN {X 0,Y 397.082,Z 106.644,A -85,B 0,C 180,E1 -11121.729,E2 -11121.729} C_VEL
LIN {X 0,Y 397.099,Z 106.642,A -85,B 0,C 180,E1 -11125.51,E2 -11125.51} C_VEL
LIN {X 0,Y 397.066,Z 106.646,A -85,B 0,C 180,E1 -11129.122,E2 -11129.122} C_VEL
LIN {X 0,Y 397.172,Z 106.635,A -85,B 0,C 180,E1 -11132.613,E2 -11132.613} C_VEL
LIN {X 0,Y 397.12,Z 106.645,A -85,B 0,C 180,E1 -11135.985,E2 -11135.985} C_VEL
LIN {X 0,Y 397.138,Z 106.638,A -85,B 0,C 180,E1 -11139.276,E2 -11139.276} C_VEL
LIN {X 0,Y 397.165,Z 106.634,A -85,B 0,C 180,E1 -11142.847,E2 -11142.847} C_VEL
LIN {X 0,Y 397.166,Z 106.639,A -85,B 0,C 180,E1 -11145.66,E2 -11145.66} C_VEL
LIN {X 0,Y 397.195,Z 106.63,A -85,B 0,C 180,E1 -11148.78,E2 -11148.78} C_VEL
LIN {X 0,Y 397.38,Z 106.609,A -85,B 0,C 180,E1 -11152.044,E2 -11152.044} C_VEL
LIN {X 0,Y 397.246,Z 106.625,A -85,B 0,C 180,E1 -11154.929,E2 -11154.929} C_VEL
LIN {X 0,Y 397.441,Z 106.601,A -85,B 0,C 180,E1 -11157.977,E2 -11157.977} C_VEL
LIN {X 0,Y 397.572,Z 106.584,A -85,B 0,C 180,E1 -11160.003,E2 -11160.003} C_VEL
LIN {X 0,Y 397.373,Z 106.612,A -85,B 0,C 180,E1 -11163.045,E2 -11163.045} C_VEL
LIN {X 0,Y 397.356,Z 106.617,A -85,B 0,C 180,E1 -11167.115,E2 -11167.115} C_VEL
LIN {X 0,Y 397.211,Z 106.628,A -85,B 0,C 180,E1 -11170.194,E2 -11170.194} C_VEL
LIN {X 0,Y 397.22,Z 106.629,A -85,B 0,C 180,E1 -11173.324,E2 -11173.324} C_VEL
LIN {X 0,Y 397.176,Z 106.635,A -85,B 0,C 180,E1 -11177.158,E2 -11177.158} C_VEL
LIN {X 0,Y 397.098,Z 106.649,A -85,B 0,C 180,E1 -11180.733,E2 -11180.733} C_VEL
LIN {X 0,Y 397.13,Z 106.639,A -85,B 0,C 180,E1 -11184.021,E2 -11184.021} C_VEL
LIN {X 0,Y 397.192,Z 106.63,A -85,B 0,C 180,E1 -11187.393,E2 -11187.393} C_VEL
LIN {X 0,Y 397.076,Z 106.647,A -85,B 0,C 180,E1 -11190.885,E2 -11190.885} C_VEL
LIN {X 0,Y 397.124,Z 106.643,A -85,B 0,C 180,E1 -11194.496,E2 -11194.496} C_VEL
LIN {X 0,Y 397.102,Z 106.647,A -85,B 0,C 180,E1 -11198.278,E2 -11198.278} C_VEL
LIN {X 0,Y 397.088,Z 106.643,A -85,B 0,C 180,E1 -11200.911,E2 -11200.911} C_VEL
LIN {X 0,Y 397.101,Z 106.645,A -85,B 0,C 180,E1 -11203.651,E2 -11203.651} C_VEL
LIN {X 0,Y 397.103,Z 106.642,A -85,B 0,C 180,E1 -11206.524,E2 -11206.524} C_VEL
LIN {X 0,Y 397.114,Z 106.641,A -85,B 0,C 180,E1 -11210.425,E2 -11210.425} C_VEL
LIN {X 0,Y 397.11,Z 106.642,A -85,B 0,C 180,E1 -11214.268,E2 -11214.268} C_VEL
LIN {X 0,Y 397.117,Z 106.642,A -85,B 0,C 180,E1 -11216.729,E2 -11216.729} C_VEL
LIN {X 0,Y 397.148,Z 106.773,A -85,B 0,C 180,E1 -11219.688,E2 -11219.688} C_VEL
LIN {X 0,Y 400.125,Z 120.203,A -85,B 0,C 180,E1 -11222.546,E2 -11222.546} C_VEL
LIN {X 0,Y 401.43,Z 127.533,A -85,B 0,C 180,E1 -11224.046,E2 -11224.046} C_VEL
LIN {X 0,Y 400.563,Z 138.989,A -85,B 0,C 180,E1 -11226.202,E2 -11226.202} C_VEL
LIN {X 0,Y 405.996,Z 171.872,A -85,B 0,C 180,E1 -11227.117,E2 -11227.117} C_VEL
LIN {X 0,Y 404.262,Z 277.392,A -85,B 0,C 180,E1 -11229.023,E2 -11229.023} C_VEL
LIN {X 0,Y 403.644,Z 291.976,A -85,B 0,C 180,E1 -11229.49,E2 -11229.49} C_VEL
LIN {X 0,Y 402.829,Z 305.386,A -85,B 0,C 180,E1 -11230.112,E2 -11230.112} C_VEL
LIN {X 0,Y 401.906,Z 319.106,A -85,B 0,C 180,E1 -11230.97,E2 -11230.97} C_VEL
LIN {X 0,Y 400.844,Z 331.987,A -85,B 0,C 180,E1 -11232.002,E2 -11232.002} C_VEL
LIN {X 0,Y 399.811,Z 343.455,A -85,B 0,C 180,E1 -11233.141,E2 -11233.141} C_VEL
LIN {X 0,Y 398.832,Z 353.978,A -85,B 0,C 180,E1 -11234.413,E2 -11234.413} C_VEL
LIN {X 0,Y 397.979,Z 364.318,A -85,B 0,C 180,E1 -11235.928,E2 -11235.928} C_VEL
LIN {X 0,Y 397.237,Z 373.063,A -85,B 0,C 180,E1 -11237.485,E2 -11237.485} C_VEL
LIN {X 0,Y 396.558,Z 381.28,A -85,B 0,C 180,E1 -11239.277,E2 -11239.277} C_VEL
LIN {X 0,Y 396.216,Z 387.062,A -85,B 0,C 180,E1 -11240.816,E2 -11240.816} C_VEL
LIN {X 0,Y 395.969,Z 391.753,A -85,B 0,C 180,E1 -11242.352,E2 -11242.352} C_VEL
LIN {X 0,Y 395.791,Z 395.637,A -85,B 0,C 180,E1 -11243.937,E2 -11243.937} C_VEL
LIN {X 0,Y 395.749,Z 399.212,A -85,B 0,C 180,E1 -11245.928,E2 -11245.928} C_VEL
LIN {X 0,Y 395.763,Z 401.475,A -85,B 0,C 180,E1 -11247.966,E2 -11247.966} C_VEL
LIN {X 0,Y 395.782,Z 402.376,A -85,B 0,C 180,E1 -11250.001,E2 -11250.001} C_VEL
LIN {X 0,Y 395.761,Z 401.937,A -85,B 0,C 180,E1 -11252.037,E2 -11252.037} C_VEL
LIN {X 0,Y 395.751,Z 400.162,A -85,B 0,C 180,E1 -11254.075,E2 -11254.075} C_VEL
LIN {X 0,Y 395.869,Z 396.928,A -85,B 0,C 180,E1 -11256.168,E2 -11256.168} C_VEL
LIN {X 0,Y 396.092,Z 392.41,A -85,B 0,C 180,E1 -11258.162,E2 -11258.162} C_VEL
LIN {X 0,Y 396.572,Z 386.162,A -85,B 0,C 180,E1 -11260.209,E2 -11260.209} C_VEL
LIN {X 0,Y 397.265,Z 379.235,A -85,B 0,C 180,E1 -11261.999,E2 -11261.999} C_VEL
LIN {X 0,Y 398.045,Z 371.506,A -85,B 0,C 180,E1 -11263.631,E2 -11263.631} C_VEL
LIN {X 0,Y 399.109,Z 361.755,A -85,B 0,C 180,E1 -11265.317,E2 -11265.317} C_VEL
LIN {X 0,Y 400.131,Z 352.929,A -85,B 0,C 180,E1 -11266.585,E2 -11266.585} C_VEL
LIN {X 0,Y 401.548,Z 341.263,A -85,B 0,C 180,E1 -11267.969,E2 -11267.969} C_VEL
LIN {X 0,Y 402.793,Z 329.616,A -85,B 0,C 180,E1 -11269.097,E2 -11269.097} C_VEL
LIN {X 0,Y 404.018,Z 317.355,A -85,B 0,C 180,E1 -11270.054,E2 -11270.054} C_VEL
LIN {X 0,Y 405.08,Z 304.654,A -85,B 0,C 180,E1 -11270.836,E2 -11270.836} C_VEL
LIN {X 0,Y 406.057,Z 290.622,A -85,B 0,C 180,E1 -11271.481,E2 -11271.481} C_VEL
LIN {X 0,Y 406.849,Z 275.7,A -85,B 0,C 180,E1 -11271.936,E2 -11271.936} C_VEL
LIN {X 0,Y 408.781,Z 171.391,A -85,B 0,C 180,E1 -11273.854,E2 -11273.854} C_VEL
LIN {X 0,Y 404.465,Z 149.255,A -85,B 0,C 180,E1 -11274.607,E2 -11274.607} C_VEL
LIN {X 0,Y 402.101,Z 138.487,A -85,B 0,C 180,E1 -11275.024,E2 -11275.024} C_VEL
LIN {X 0,Y 402.805,Z 131.369,A -85,B 0,C 180,E1 -11276.419,E2 -11276.419} C_VEL
LIN {X 0,Y 400.522,Z 119.954,A -85,B 0,C 180,E1 -11278.98,E2 -11278.98} C_VEL
LIN {X 0,Y 397.904,Z 109.806,A -85,B 0,C 180,E1 -11281.404,E2 -11281.404} C_VEL
LIN {X 0,Y 397.108,Z 106.646,A -85,B 0,C 180,E1 -11282.22,E2 -11282.22} C_VEL
LIN {X 0,Y 397.108,Z 106.648,A -85,B 0,C 180,E1 -11285.736,E2 -11285.736} C_VEL
LIN {X 0,Y 397.113,Z 106.645,A -85,B 0,C 180,E1 -11288.856,E2 -11288.856} C_VEL
LIN {X 0,Y 397.078,Z 106.65,A -85,B 0,C 180,E1 -11292.268,E2 -11292.268} C_VEL
LIN {X 0,Y 397.101,Z 106.644,A -85,B 0,C 180,E1 -11295.068,E2 -11295.068} C_VEL
LIN {X 0,Y 397.077,Z 106.635,A -85,B 0,C 180,E1 -11298.021,E2 -11298.021} C_VEL
LIN {X 0,Y 397.114,Z 106.643,A -85,B 0,C 180,E1 -11301.143,E2 -11301.143} C_VEL
LIN {X 0,Y 397.113,Z 106.642,A -85,B 0,C 180,E1 -11304.5,E2 -11304.5} C_VEL
LIN {X 0,Y 397.092,Z 106.644,A -85,B 0,C 180,E1 -11307.927,E2 -11307.927} C_VEL
LIN {X 0,Y 397.132,Z 106.64,A -85,B 0,C 180,E1 -11310.294,E2 -11310.294} C_VEL
LIN {X 0,Y 397.109,Z 106.644,A -85,B 0,C 180,E1 -11313.737,E2 -11313.737} C_VEL
LIN {X 0,Y 397.118,Z 106.642,A -85,B 0,C 180,E1 -11317.083,E2 -11317.083} C_VEL
LIN {X 0,Y 397.16,Z 106.63,A -85,B 0,C 180,E1 -11320.351,E2 -11320.351} C_VEL
LIN {X 0,Y 397.179,Z 106.628,A -85,B 0,C 180,E1 -11323.551,E2 -11323.551} C_VEL
LIN {X 0,Y 397.241,Z 106.628,A -85,B 0,C 180,E1 -11326.7,E2 -11326.7} C_VEL
LIN {X 0,Y 397.227,Z 106.627,A -85,B 0,C 180,E1 -11329.806,E2 -11329.806} C_VEL
LIN {X 0,Y 397.305,Z 106.615,A -85,B 0,C 180,E1 -11332.884,E2 -11332.884} C_VEL
LIN {X 0,Y 397.25,Z 106.626,A -85,B 0,C 180,E1 -11334.922,E2 -11334.922} C_VEL
LIN {X 0,Y 397.454,Z 106.597,A -85,B 0,C 180,E1 -11337.97,E2 -11337.97} C_VEL
LIN {X 0,Y 397.582,Z 106.585,A -85,B 0,C 180,E1 -11339.997,E2 -11339.997} C_VEL
LIN {X 0,Y 397.374,Z 106.609,A -85,B 0,C 180,E1 -11343.038,E2 -11343.038} C_VEL
LIN {X 0,Y 397.323,Z 106.613,A -85,B 0,C 180,E1 -11346.509,E2 -11346.509} C_VEL
LIN {X 0,Y 397.239,Z 106.623,A -85,B 0,C 180,E1 -11349.158,E2 -11349.158} C_VEL
LIN {X 0,Y 397.221,Z 106.626,A -85,B 0,C 180,E1 -11352.254,E2 -11352.254} C_VEL
LIN {X 0,Y 397.179,Z 106.638,A -85,B 0,C 180,E1 -11355.388,E2 -11355.388} C_VEL
LIN {X 0,Y 397.159,Z 106.637,A -85,B 0,C 180,E1 -11358.569,E2 -11358.569} C_VEL
LIN {X 0,Y 397.104,Z 106.645,A -85,B 0,C 180,E1 -11361.814,E2 -11361.814} C_VEL
LIN {X 0,Y 397.145,Z 106.637,A -85,B 0,C 180,E1 -11365.507,E2 -11365.507} C_VEL
LIN {X 0,Y 397.109,Z 106.641,A -85,B 0,C 180,E1 -11368.54,E2 -11368.54} C_VEL
LIN {X 0,Y 397.068,Z 106.649,A -85,B 0,C 180,E1 -11372.067,E2 -11372.067} C_VEL
LIN {X 0,Y 397.106,Z 106.646,A -85,B 0,C 180,E1 -11375.499,E2 -11375.499} C_VEL
LIN {X 0,Y 397.112,Z 106.643,A -85,B 0,C 180,E1 -11378.856,E2 -11378.856} C_VEL
LIN {X 0,Y 397.052,Z 106.654,A -85,B 0,C 180,E1 -11382.263,E2 -11382.263} C_VEL
LIN {X 0,Y 397.098,Z 106.688,A -85,B 0,C 180,E1 -11385.466,E2 -11385.466} C_VEL
LIN {X 0,Y 400.066,Z 119.061,A -85,B 0,C 180,E1 -11388.711,E2 -11388.711} C_VEL
LIN {X 0,Y 400.217,Z 119.83,A -85,B 0,C 180,E1 -11388.899,E2 -11388.899} C_VEL
LIN {X 0,Y 406.748,Z 135.293,A -85,B 0,C 180,E1 -11389.712,E2 -11389.712} C_VEL
LIN {X 0,Y 409.296,Z 146.437,A -85,B 0,C 180,E1 -11390.12,E2 -11390.12} C_VEL
LIN {X 0,Y 407.108,Z 256.537,A -85,B 0,C 180,E1 -11392.145,E2 -11392.145} C_VEL
LIN {X 0,Y 406.449,Z 271.071,A -85,B 0,C 180,E1 -11392.616,E2 -11392.616} C_VEL
LIN {X 0,Y 405.573,Z 285.099,A -85,B 0,C 180,E1 -11393.283,E2 -11393.283} C_VEL
LIN {X 0,Y 404.571,Z 298.016,A -85,B 0,C 180,E1 -11394.105,E2 -11394.105} C_VEL
LIN {X 0,Y 403.483,Z 309.782,A -85,B 0,C 180,E1 -11395.051,E2 -11395.051} C_VEL
LIN {X 0,Y 402.275,Z 321.015,A -85,B 0,C 180,E1 -11396.159,E2 -11396.159} C_VEL
LIN {X 0,Y 401,Z 332.155,A -85,B 0,C 180,E1 -11397.501,E2 -11397.501} C_VEL
LIN {X 0,Y 399.733,Z 342.677,A -85,B 0,C 180,E1 -11399.05,E2 -11399.05} C_VEL
LIN {X 0,Y 398.593,Z 351.847,A -85,B 0,C 180,E1 -11400.705,E2 -11400.705} C_VEL
LIN {X 0,Y 397.734,Z 359.203,A -85,B 0,C 180,E1 -11402.327,E2 -11402.327} C_VEL
LIN {X 0,Y 396.969,Z 366.082,A -85,B 0,C 180,E1 -11404.209,E2 -11404.209} C_VEL
LIN {X 0,Y 396.489,Z 371.104,A -85,B 0,C 180,E1 -11405.939,E2 -11405.939} C_VEL
LIN {X 0,Y 396.227,Z 374.126,A -85,B 0,C 180,E1 -11407.257,E2 -11407.257} C_VEL
LIN {X 0,Y 395.869,Z 377.519,A -85,B 0,C 180,E1 -11409.201,E2 -11409.201} C_VEL
LIN {X 0,Y 395.679,Z 379.814,A -85,B 0,C 180,E1 -11411.353,E2 -11411.353} C_VEL
LIN {X 0,Y 395.603,Z 380.655,A -85,B 0,C 180,E1 -11413.584,E2 -11413.584} C_VEL
LIN {X 0,Y 395.583,Z 380.045,A -85,B 0,C 180,E1 -11415.596,E2 -11415.596} C_VEL
LIN {X 0,Y 395.725,Z 378.015,A -85,B 0,C 180,E1 -11417.693,E2 -11417.693} C_VEL
LIN {X 0,Y 395.921,Z 374.551,A -85,B 0,C 180,E1 -11419.774,E2 -11419.774} C_VEL
LIN {X 0,Y 396.226,Z 369.581,A -85,B 0,C 180,E1 -11421.841,E2 -11421.841} C_VEL
LIN {X 0,Y 396.633,Z 364.574,A -85,B 0,C 180,E1 -11423.442,E2 -11423.442} C_VEL
LIN {X 0,Y 397.111,Z 357.855,A -85,B 0,C 180,E1 -11425.176,E2 -11425.176} C_VEL
LIN {X 0,Y 397.916,Z 349.269,A -85,B 0,C 180,E1 -11426.961,E2 -11426.961} C_VEL
LIN {X 0,Y 398.743,Z 340.32,A -85,B 0,C 180,E1 -11428.484,E2 -11428.484} C_VEL
LIN {X 0,Y 399.159,Z 336.081,A -85,B 0,C 180,E1 -11429.112,E2 -11429.112} C_VEL
LIN {X 0,Y 398.888,Z 331.91,A -85,B 0,C 180,E1 -11429.71,E2 -11429.71} C_VEL
LIN {X 0,Y 396.689,Z 324.925,A -85,B 0,C 180,E1 -11430.681,E2 -11430.681} C_VEL
LIN {X 0,Y 394.541,Z 317.634,A -85,B 0,C 180,E1 -11431.596,E2 -11431.596} C_VEL
LIN {X 0,Y 394.342,Z 312.797,A -85,B 0,C 180,E1 -11432.099,E2 -11432.099} C_VEL
LIN {X 0,Y 395.511,Z 299.972,A -85,B 0,C 180,E1 -11433.182,E2 -11433.182} C_VEL
LIN {X 0,Y 396.329,Z 286.707,A -85,B 0,C 180,E1 -11434.066,E2 -11434.066} C_VEL
LIN {X 0,Y 397.027,Z 272.902,A -85,B 0,C 180,E1 -11434.758,E2 -11434.758} C_VEL
LIN {X 0,Y 397.547,Z 258.486,A -85,B 0,C 180,E1 -11435.26,E2 -11435.26} C_VEL
LIN {X 0,Y 398.029,Z 236.756,A -85,B 0,C 180,E1 -11435.699,E2 -11435.699} C_VEL
LIN {X 0,Y 399.569,Z 146.387,A -85,B 0,C 180,E1 -11437.333,E2 -11437.333} C_VEL
LIN {X 0,Y 395.868,Z 128.651,A -85,B 0,C 180,E1 -11437.873,E2 -11437.873} C_VEL
LIN {X 0,Y 392.624,Z 119.482,A -85,B 0,C 180,E1 -11438.232,E2 -11438.232} C_VEL
LIN {X 0,Y 390.164,Z 107.514,A -85,B 0,C 180,E1 -11441.098,E2 -11441.098} C_VEL
LIN {X 0,Y 390.185,Z 107.511,A -85,B 0,C 180,E1 -11443.54,E2 -11443.54} C_VEL
LIN {X 0,Y 390.146,Z 107.512,A -85,B 0,C 180,E1 -11447.324,E2 -11447.324} C_VEL
LIN {X 0,Y 390.073,Z 107.52,A -85,B 0,C 180,E1 -11451.12,E2 -11451.12} C_VEL
LIN {X 0,Y 390.049,Z 107.52,A -85,B 0,C 180,E1 -11454.481,E2 -11454.481} C_VEL
LIN {X 0,Y 390.08,Z 107.517,A -85,B 0,C 180,E1 -11458.026,E2 -11458.026} C_VEL
LIN {X 0,Y 390.014,Z 107.528,A -85,B 0,C 180,E1 -11461.503,E2 -11461.503} C_VEL
LIN {X 0,Y 390.058,Z 107.524,A -85,B 0,C 180,E1 -11465.208,E2 -11465.208} C_VEL
LIN {X 0,Y 390.08,Z 107.517,A -85,B 0,C 180,E1 -11467.774,E2 -11467.774} C_VEL
LIN {X 0,Y 390.061,Z 107.525,A -85,B 0,C 180,E1 -11470.83,E2 -11470.83} C_VEL
LIN {X 0,Y 390.103,Z 107.513,A -85,B 0,C 180,E1 -11473.901,E2 -11473.901} C_VEL
LIN {X 0,Y 390.089,Z 107.521,A -85,B 0,C 180,E1 -11476.801,E2 -11476.801} C_VEL
LIN {X 0,Y 390.05,Z 107.52,A -85,B 0,C 180,E1 -11479.566,E2 -11479.566} C_VEL
LIN {X 0,Y 390.02,Z 107.53,A -85,B 0,C 180,E1 -11482.451,E2 -11482.451} C_VEL
LIN {X 0,Y 390.041,Z 107.524,A -85,B 0,C 180,E1 -11486.048,E2 -11486.048} C_VEL
LIN {X 0,Y 390.024,Z 107.528,A -85,B 0,C 180,E1 -11488.501,E2 -11488.501} C_VEL
LIN {X 0,Y 390.093,Z 107.52,A -85,B 0,C 180,E1 -11492.073,E2 -11492.073} C_VEL
LIN {X 0,Y 390.064,Z 107.519,A -85,B 0,C 180,E1 -11495.523,E2 -11495.523} C_VEL
LIN {X 0,Y 390.09,Z 107.515,A -85,B 0,C 180,E1 -11498.884,E2 -11498.884} C_VEL
LIN {X 0,Y 390.131,Z 107.51,A -85,B 0,C 180,E1 -11502.695,E2 -11502.695} C_VEL
LIN {X 0,Y 390.177,Z 107.504,A -85,B 0,C 180,E1 -11506.565,E2 -11506.565} C_VEL
LIN {X 0,Y 390.164,Z 107.512,A -85,B 0,C 180,E1 -11509.627,E2 -11509.627} C_VEL
LIN {X 0,Y 390.305,Z 107.489,A -85,B 0,C 180,E1 -11512.763,E2 -11512.763} C_VEL
LIN {X 0,Y 390.218,Z 107.5,A -85,B 0,C 180,E1 -11514.837,E2 -11514.837} C_VEL
LIN {X 0,Y 390.41,Z 107.477,A -85,B 0,C 180,E1 -11517.94,E2 -11517.94} C_VEL
LIN {X 0,Y 390.541,Z 107.46,A -85,B 0,C 180,E1 -11520.003,E2 -11520.003} C_VEL
LIN {X 0,Y 390.307,Z 107.493,A -85,B 0,C 180,E1 -11523.1,E2 -11523.1} C_VEL
LIN {X 0,Y 390.321,Z 107.486,A -85,B 0,C 180,E1 -11526.205,E2 -11526.205} C_VEL
LIN {X 0,Y 390.306,Z 107.488,A -85,B 0,C 180,E1 -11528.285,E2 -11528.285} C_VEL
LIN {X 0,Y 390.164,Z 107.508,A -85,B 0,C 180,E1 -11532.486,E2 -11532.486} C_VEL
LIN {X 0,Y 390.133,Z 107.51,A -85,B 0,C 180,E1 -11535.68,E2 -11535.68} C_VEL
LIN {X 0,Y 390.101,Z 107.519,A -85,B 0,C 180,E1 -11538.925,E2 -11538.925} C_VEL
LIN {X 0,Y 390.036,Z 107.524,A -85,B 0,C 180,E1 -11542.237,E2 -11542.237} C_VEL
LIN {X 0,Y 390.116,Z 107.512,A -85,B 0,C 180,E1 -11545.746,E2 -11545.746} C_VEL
LIN {X 0,Y 390.056,Z 107.52,A -85,B 0,C 180,E1 -11549.112,E2 -11549.112} C_VEL
LIN {X 0,Y 390.041,Z 107.524,A -85,B 0,C 180,E1 -11552.724,E2 -11552.724} C_VEL
LIN {X 0,Y 390.055,Z 107.522,A -85,B 0,C 180,E1 -11555.828,E2 -11555.828} C_VEL
LIN {X 0,Y 390.069,Z 107.518,A -85,B 0,C 180,E1 -11559.221,E2 -11559.221} C_VEL
LIN {X 0,Y 390.043,Z 107.524,A -85,B 0,C 180,E1 -11562.377,E2 -11562.377} C_VEL
LIN {X 0,Y 390.045,Z 107.522,A -85,B 0,C 180,E1 -11565.357,E2 -11565.357} C_VEL
LIN {X 0,Y 390.032,Z 107.525,A -85,B 0,C 180,E1 -11568.189,E2 -11568.189} C_VEL
LIN {X 0,Y 390.088,Z 107.515,A -85,B 0,C 180,E1 -11570.91,E2 -11570.91} C_VEL
LIN {X 0,Y 390.087,Z 107.516,A -85,B 0,C 180,E1 -11574.795,E2 -11574.795} C_VEL
LIN {X 0,Y 390.031,Z 107.527,A -85,B 0,C 180,E1 -11578.498,E2 -11578.498} C_VEL
LIN {X 0,Y 390.103,Z 107.585,A -85,B 0,C 180,E1 -11579.371,E2 -11579.371} C_VEL
LIN {X 0,Y 393.341,Z 122.293,A -85,B 0,C 180,E1 -11582.559,E2 -11582.559} C_VEL
LIN {X 0,Y 394.476,Z 128.418,A -85,B 0,C 180,E1 -11583.837,E2 -11583.837} C_VEL
LIN {X 0,Y 393.728,Z 138.861,A -85,B 0,C 180,E1 -11585.842,E2 -11585.842} C_VEL
LIN {X 0,Y 399.322,Z 172.507,A -85,B 0,C 180,E1 -11586.789,E2 -11586.789} C_VEL
LIN {X 0,Y 397.505,Z 277.454,A -85,B 0,C 180,E1 -11588.717,E2 -11588.717} C_VEL
LIN {X 0,Y 396.866,Z 291.952,A -85,B 0,C 180,E1 -11589.191,E2 -11589.191} C_VEL
LIN {X 0,Y 395.963,Z 306.459,A -85,B 0,C 180,E1 -11589.888,E2 -11589.888} C_VEL
LIN {X 0,Y 394.992,Z 320.016,A -85,B 0,C 180,E1 -11590.767,E2 -11590.767} C_VEL
LIN {X 0,Y 393.907,Z 332.593,A -85,B 0,C 180,E1 -11591.808,E2 -11591.808} C_VEL
LIN {X 0,Y 392.845,Z 343.92,A -85,B 0,C 180,E1 -11592.967,E2 -11592.967} C_VEL
LIN {X 0,Y 391.757,Z 355.281,A -85,B 0,C 180,E1 -11594.391,E2 -11594.391} C_VEL
LIN {X 0,Y 390.871,Z 365.341,A -85,B 0,C 180,E1 -11595.936,E2 -11595.936} C_VEL
LIN {X 0,Y 390.114,Z 373.866,A -85,B 0,C 180,E1 -11597.517,E2 -11597.517} C_VEL
LIN {X 0,Y 389.462,Z 381.902,A -85,B 0,C 180,E1 -11599.342,E2 -11599.342} C_VEL
LIN {X 0,Y 389.059,Z 388.358,A -85,B 0,C 180,E1 -11601.169,E2 -11601.169} C_VEL
LIN {X 0,Y 388.769,Z 394.06,A -85,B 0,C 180,E1 -11603.253,E2 -11603.253} C_VEL
LIN {X 0,Y 388.678,Z 397.272,A -85,B 0,C 180,E1 -11604.814,E2 -11604.814} C_VEL
LIN {X 0,Y 388.625,Z 400.266,A -85,B 0,C 180,E1 -11606.892,E2 -11606.892} C_VEL
LIN {X 0,Y 388.705,Z 401.875,A -85,B 0,C 180,E1 -11608.965,E2 -11608.965} C_VEL
LIN {X 0,Y 388.705,Z 402.135,A -85,B 0,C 180,E1 -11611.037,E2 -11611.037} C_VEL
LIN {X 0,Y 388.623,Z 401.058,A -85,B 0,C 180,E1 -11613.111,E2 -11613.111} C_VEL
LIN {X 0,Y 388.698,Z 398.639,A -85,B 0,C 180,E1 -11615.188,E2 -11615.188} C_VEL
LIN {X 0,Y 388.87,Z 394.819,A -85,B 0,C 180,E1 -11617.269,E2 -11617.269} C_VEL
LIN {X 0,Y 389.268,Z 389.47,A -85,B 0,C 180,E1 -11619.353,E2 -11619.353} C_VEL
LIN {X 0,Y 389.678,Z 384.344,A -85,B 0,C 180,E1 -11620.918,E2 -11620.918} C_VEL
LIN {X 0,Y 390.584,Z 377.042,A -85,B 0,C 180,E1 -11622.735,E2 -11622.735} C_VEL
LIN {X 0,Y 391.494,Z 368.02,A -85,B 0,C 180,E1 -11624.557,E2 -11624.557} C_VEL
LIN {X 0,Y 392.665,Z 358.59,A -85,B 0,C 180,E1 -11626.108,E2 -11626.108} C_VEL
LIN {X 0,Y 393.961,Z 348.179,A -85,B 0,C 180,E1 -11627.521,E2 -11627.521} C_VEL
LIN {X 0,Y 395.398,Z 336.719,A -85,B 0,C 180,E1 -11628.795,E2 -11628.795} C_VEL
LIN {X 0,Y 396.781,Z 323.92,A -85,B 0,C 180,E1 -11629.95,E2 -11629.95} C_VEL
LIN {X 0,Y 397.927,Z 311.785,A -85,B 0,C 180,E1 -11630.822,E2 -11630.822} C_VEL
LIN {X 0,Y 399.036,Z 298.218,A -85,B 0,C 180,E1 -11631.573,E2 -11631.573} C_VEL
LIN {X 0,Y 399.969,Z 285.063,A -85,B 0,C 180,E1 -11632.096,E2 -11632.096} C_VEL
LIN {X 0,Y 400.582,Z 270.908,A -85,B 0,C 180,E1 -11632.468,E2 -11632.468} C_VEL
LIN {X 0,Y 402.507,Z 173.286,A -85,B 0,C 180,E1 -11634.274,E2 -11634.274} C_VEL
LIN {X 0,Y 398.849,Z 153.494,A -85,B 0,C 180,E1 -11634.948,E2 -11634.948} C_VEL
LIN {X 0,Y 395.502,Z 138.229,A -85,B 0,C 180,E1 -11635.556,E2 -11635.556} C_VEL
LIN {X 0,Y 395.994,Z 133.141,A -85,B 0,C 180,E1 -11636.574,E2 -11636.574} C_VEL
LIN {X 0,Y 393.867,Z 122.415,A -85,B 0,C 180,E1 -11639.03,E2 -11639.03} C_VEL
LIN {X 0,Y 391.077,Z 111.546,A -85,B 0,C 180,E1 -11641.681,E2 -11641.681} C_VEL
LIN {X 0,Y 390.082,Z 107.521,A -85,B 0,C 180,E1 -11642.719,E2 -11642.719} C_VEL
LIN {X 0,Y 390.057,Z 107.527,A -85,B 0,C 180,E1 -11645.822,E2 -11645.822} C_VEL
LIN {X 0,Y 390.056,Z 107.524,A -85,B 0,C 180,E1 -11649.213,E2 -11649.213} C_VEL
LIN {X 0,Y 390.053,Z 107.524,A -85,B 0,C 180,E1 -11652.373,E2 -11652.373} C_VEL
LIN {X 0,Y 390.058,Z 107.521,A -85,B 0,C 180,E1 -11655.354,E2 -11655.354} C_VEL
LIN {X 0,Y 390.04,Z 107.509,A -85,B 0,C 180,E1 -11658.185,E2 -11658.185} C_VEL
LIN {X 0,Y 390.077,Z 107.518,A -85,B 0,C 180,E1 -11660.903,E2 -11660.903} C_VEL
LIN {X 0,Y 390.084,Z 107.518,A -85,B 0,C 180,E1 -11664.79,E2 -11664.79} C_VEL
LIN {X 0,Y 390.037,Z 107.521,A -85,B 0,C 180,E1 -11668.494,E2 -11668.494} C_VEL
LIN {X 0,Y 390.052,Z 107.516,A -85,B 0,C 180,E1 -11672.062,E2 -11672.062} C_VEL
LIN {X 0,Y 390.074,Z 107.513,A -85,B 0,C 180,E1 -11675.516,E2 -11675.516} C_VEL
LIN {X 0,Y 390.069,Z 107.52,A -85,B 0,C 180,E1 -11678.876,E2 -11678.876} C_VEL
LIN {X 0,Y 390.139,Z 107.512,A -85,B 0,C 180,E1 -11682.164,E2 -11682.164} C_VEL
LIN {X 0,Y 390.156,Z 107.509,A -85,B 0,C 180,E1 -11685.39,E2 -11685.39} C_VEL
LIN {X 0,Y 390.158,Z 107.504,A -85,B 0,C 180,E1 -11688.568,E2 -11688.568} C_VEL
LIN {X 0,Y 390.267,Z 107.492,A -85,B 0,C 180,E1 -11692.083,E2 -11692.083} C_VEL
LIN {X 0,Y 390.22,Z 107.502,A -85,B 0,C 180,E1 -11694.83,E2 -11694.83} C_VEL
LIN {X 0,Y 390.422,Z 107.472,A -85,B 0,C 180,E1 -11697.933,E2 -11697.933} C_VEL
LIN {X 0,Y 390.552,Z 107.46,A -85,B 0,C 180,E1 -11699.997,E2 -11699.997} C_VEL
LIN {X 0,Y 390.308,Z 107.49,A -85,B 0,C 180,E1 -11703.093,E2 -11703.093} C_VEL
LIN {X 0,Y 390.281,Z 107.491,A -85,B 0,C 180,E1 -11706.501,E2 -11706.501} C_VEL
LIN {X 0,Y 390.197,Z 107.5,A -85,B 0,C 180,E1 -11709.325,E2 -11709.325} C_VEL
LIN {X 0,Y 390.173,Z 107.503,A -85,B 0,C 180,E1 -11712.479,E2 -11712.479} C_VEL
LIN {X 0,Y 390.139,Z 107.512,A -85,B 0,C 180,E1 -11715.673,E2 -11715.673} C_VEL
LIN {X 0,Y 390.103,Z 107.517,A -85,B 0,C 180,E1 -11718.918,E2 -11718.918} C_VEL
LIN {X 0,Y 390.041,Z 107.523,A -85,B 0,C 180,E1 -11722.23,E2 -11722.23} C_VEL
LIN {X 0,Y 390.112,Z 107.511,A -85,B 0,C 180,E1 -11725.738,E2 -11725.738} C_VEL
LIN {X 0,Y 390.045,Z 107.512,A -85,B 0,C 180,E1 -11729.106,E2 -11729.106} C_VEL
LIN {X 0,Y 390.032,Z 107.526,A -85,B 0,C 180,E1 -11732.717,E2 -11732.717} C_VEL
LIN {X 0,Y 390.043,Z 107.526,A -85,B 0,C 180,E1 -11735.821,E2 -11735.821} C_VEL
LIN {X 0,Y 390.053,Z 107.526,A -85,B 0,C 180,E1 -11739.213,E2 -11739.213} C_VEL
LIN {X 0,Y 390.026,Z 107.529,A -85,B 0,C 180,E1 -11742.37,E2 -11742.37} C_VEL
LIN {X 0,Y 390.028,Z 107.535,A -85,B 0,C 180,E1 -11744.955,E2 -11744.955} C_VEL
LIN {X 0,Y 393.067,Z 120.001,A -85,B 0,C 180,E1 -11748.316,E2 -11748.316} C_VEL
LIN {X 0,Y 400.744,Z 137.736,A -85,B 0,C 180,E1 -11749.304,E2 -11749.304} C_VEL
LIN {X 0,Y 402.989,Z 147.591,A -85,B 0,C 180,E1 -11749.674,E2 -11749.674} C_VEL
LIN {X 0,Y 400.738,Z 256.03,A -85,B 0,C 180,E1 -11751.694,E2 -11751.694} C_VEL
LIN {X 0,Y 400.055,Z 270.68,A -85,B 0,C 180,E1 -11752.165,E2 -11752.165} C_VEL
LIN {X 0,Y 399.198,Z 284.298,A -85,B 0,C 180,E1 -11752.812,E2 -11752.812} C_VEL
LIN {X 0,Y 398.176,Z 296.724,A -85,B 0,C 180,E1 -11753.593,E2 -11753.593} C_VEL
LIN {X 0,Y 397.101,Z 308.092,A -85,B 0,C 180,E1 -11754.492,E2 -11754.492} C_VEL
LIN {X 0,Y 395.738,Z 320.196,A -85,B 0,C 180,E1 -11755.676,E2 -11755.676} C_VEL
LIN {X 0,Y 394.471,Z 330.87,A -85,B 0,C 180,E1 -11756.956,E2 -11756.956} C_VEL
LIN {X 0,Y 393.115,Z 341.283,A -85,B 0,C 180,E1 -11758.47,E2 -11758.47} C_VEL
LIN {X 0,Y 391.873,Z 350.738,A -85,B 0,C 180,E1 -11760.152,E2 -11760.152} C_VEL
LIN {X 0,Y 390.957,Z 358.028,A -85,B 0,C 180,E1 -11761.733,E2 -11761.733} C_VEL
LIN {X 0,Y 390.289,Z 363.821,A -85,B 0,C 180,E1 -11763.243,E2 -11763.243} C_VEL
LIN {X 0,Y 389.677,Z 369.124,A -85,B 0,C 180,E1 -11764.922,E2 -11764.922} C_VEL
LIN {X 0,Y 389.194,Z 374.273,A -85,B 0,C 180,E1 -11767.052,E2 -11767.052} C_VEL
LIN {X 0,Y 388.841,Z 377.372,A -85,B 0,C 180,E1 -11768.807,E2 -11768.807} C_VEL
LIN {X 0,Y 388.622,Z 379.823,A -85,B 0,C 180,E1 -11771.002,E2 -11771.002} C_VEL
LIN {X 0,Y 388.515,Z 380.802,A -85,B 0,C 180,E1 -11773.175,E2 -11773.175} C_VEL
LIN {X 0,Y 388.479,Z 380.359,A -85,B 0,C 180,E1 -11775.327,E2 -11775.327} C_VEL
LIN {X 0,Y 388.621,Z 378.425,A -85,B 0,C 180,E1 -11777.545,E2 -11777.545} C_VEL
LIN {X 0,Y 388.806,Z 375.24,A -85,B 0,C 180,E1 -11779.585,E2 -11779.585} C_VEL
LIN {X 0,Y 389.129,Z 370.43,A -85,B 0,C 180,E1 -11781.691,E2 -11781.691} C_VEL
LIN {X 0,Y 389.47,Z 365.937,A -85,B 0,C 180,E1 -11783.217,E2 -11783.217} C_VEL
LIN {X 0,Y 390.001,Z 359.061,A -85,B 0,C 180,E1 -11785.088,E2 -11785.088} C_VEL
LIN {X 0,Y 390.796,Z 350.684,A -85,B 0,C 180,E1 -11786.906,E2 -11786.906} C_VEL
LIN {X 0,Y 391.62,Z 341.975,A -85,B 0,C 180,E1 -11788.456,E2 -11788.456} C_VEL
LIN {X 0,Y 392.667,Z 331.427,A -85,B 0,C 180,E1 -11789.999,E2 -11789.999} C_VEL
LIN {X 0,Y 393.757,Z 320.359,A -85,B 0,C 180,E1 -11791.324,E2 -11791.324} C_VEL
LIN {X 0,Y 394.342,Z 312.797,A -85,B 0,C 180,E1 -11792.099,E2 -11792.099} C_VEL
LIN {X 0,Y 394.149,Z 307.888,A -85,B 0,C 180,E1 -11792.578,E2 -11792.578} C_VEL
LIN {X 0,Y 392.039,Z 299.796,A -85,B 0,C 180,E1 -11793.359,E2 -11793.359} C_VEL
LIN {X 0,Y 389.881,Z 291.398,A -85,B 0,C 180,E1 -11794.065,E2 -11794.065} C_VEL
LIN {X 0,Y 389.601,Z 286.012,A -85,B 0,C 180,E1 -11794.42,E2 -11794.42} C_VEL
LIN {X 0,Y 390.369,Z 271.678,A -85,B 0,C 180,E1 -11795.131,E2 -11795.131} C_VEL
LIN {X 0,Y 390.841,Z 257.715,A -85,B 0,C 180,E1 -11795.61,E2 -11795.61} C_VEL
LIN {X 0,Y 391.498,Z 224.624,A -85,B 0,C 180,E1 -11796.256,E2 -11796.256} C_VEL
LIN {X 0,Y 392.848,Z 146.921,A -85,B 0,C 180,E1 -11797.686,E2 -11797.686} C_VEL
LIN {X 0,Y 389.355,Z 130.579,A -85,B 0,C 180,E1 -11798.197,E2 -11798.197} C_VEL
LIN {X 0,Y 385.46,Z 119.589,A -85,B 0,C 180,E1 -11798.651,E2 -11798.651} C_VEL
LIN {X 0,Y 383.105,Z 108.395,A -85,B 0,C 180,E1 -11801.439,E2 -11801.439} C_VEL
LIN {X 0,Y 383.096,Z 108.387,A -85,B 0,C 180,E1 -11804.881,E2 -11804.881} C_VEL
LIN {X 0,Y 383.066,Z 108.391,A -85,B 0,C 180,E1 -11808.172,E2 -11808.172} C_VEL
LIN {X 0,Y 383.039,Z 108.4,A -85,B 0,C 180,E1 -11811.526,E2 -11811.526} C_VEL
LIN {X 0,Y 383.019,Z 108.398,A -85,B 0,C 180,E1 -11814.961,E2 -11814.961} C_VEL
LIN {X 0,Y 383.014,Z 108.397,A -85,B 0,C 180,E1 -11818.493,E2 -11818.493} C_VEL
LIN {X 0,Y 382.974,Z 108.402,A -85,B 0,C 180,E1 -11822.429,E2 -11822.429} C_VEL
LIN {X 0,Y 383.008,Z 108.397,A -85,B 0,C 180,E1 -11825.955,E2 -11825.955} C_VEL
LIN {X 0,Y 383.032,Z 108.397,A -85,B 0,C 180,E1 -11828.595,E2 -11828.595} C_VEL
LIN {X 0,Y 383.018,Z 108.398,A -85,B 0,C 180,E1 -11831.341,E2 -11831.341} C_VEL
LIN {X 0,Y 383.053,Z 108.394,A -85,B 0,C 180,E1 -11834.319,E2 -11834.319} C_VEL
LIN {X 0,Y 383.045,Z 108.394,A -85,B 0,C 180,E1 -11837.252,E2 -11837.252} C_VEL
LIN {X 0,Y 382.994,Z 108.404,A -85,B 0,C 180,E1 -11840.414,E2 -11840.414} C_VEL
LIN {X 0,Y 382.999,Z 108.401,A -85,B 0,C 180,E1 -11844.047,E2 -11844.047} C_VEL
LIN {X 0,Y 383.011,Z 108.399,A -85,B 0,C 180,E1 -11847.856,E2 -11847.856} C_VEL
LIN {X 0,Y 383.04,Z 108.395,A -85,B 0,C 180,E1 -11851.723,E2 -11851.723} C_VEL
LIN {X 0,Y 383.034,Z 108.394,A -85,B 0,C 180,E1 -11855.043,E2 -11855.043} C_VEL
LIN {X 0,Y 383.056,Z 108.393,A -85,B 0,C 180,E1 -11858.477,E2 -11858.477} C_VEL
LIN {X 0,Y 383.077,Z 108.394,A -85,B 0,C 180,E1 -11861.831,E2 -11861.831} C_VEL
LIN {X 0,Y 383.097,Z 108.387,A -85,B 0,C 180,E1 -11865.122,E2 -11865.122} C_VEL
LIN {X 0,Y 383.092,Z 108.388,A -85,B 0,C 180,E1 -11868.362,E2 -11868.362} C_VEL
LIN {X 0,Y 383.289,Z 108.365,A -85,B 0,C 180,E1 -11871.936,E2 -11871.936} C_VEL
LIN {X 0,Y 383.19,Z 108.375,A -85,B 0,C 180,E1 -11874.742,E2 -11874.742} C_VEL
LIN {X 0,Y 383.377,Z 108.353,A -85,B 0,C 180,E1 -11877.902,E2 -11877.902} C_VEL
LIN {X 0,Y 383.51,Z 108.335,A -85,B 0,C 180,E1 -11880.003,E2 -11880.003} C_VEL
LIN {X 0,Y 383.243,Z 108.374,A -85,B 0,C 180,E1 -11883.157,E2 -11883.157} C_VEL
LIN {X 0,Y 383.279,Z 108.364,A -85,B 0,C 180,E1 -11886.32,E2 -11886.32} C_VEL
LIN {X 0,Y 383.252,Z 108.368,A -85,B 0,C 180,E1 -11888.439,E2 -11888.439} C_VEL
LIN {X 0,Y 383.09,Z 108.388,A -85,B 0,C 180,E1 -11891.645,E2 -11891.645} C_VEL
LIN {X 0,Y 383.104,Z 108.392,A -85,B 0,C 180,E1 -11894.885,E2 -11894.885} C_VEL
LIN {X 0,Y 383.084,Z 108.389,A -85,B 0,C 180,E1 -11898.175,E2 -11898.175} C_VEL
LIN {X 0,Y 382.989,Z 108.4,A -85,B 0,C 180,E1 -11901.534,E2 -11901.534} C_VEL
LIN {X 0,Y 383.049,Z 108.395,A -85,B 0,C 180,E1 -11904.963,E2 -11904.963} C_VEL
LIN {X 0,Y 383.038,Z 108.4,A -85,B 0,C 180,E1 -11908.496,E2 -11908.496} C_VEL
LIN {X 0,Y 383.007,Z 108.402,A -85,B 0,C 180,E1 -11912.153,E2 -11912.153} C_VEL
LIN {X 0,Y 383.017,Z 108.399,A -85,B 0,C 180,E1 -11914.671,E2 -11914.671} C_VEL
LIN {X 0,Y 382.999,Z 108.402,A -85,B 0,C 180,E1 -11917.906,E2 -11917.906} C_VEL
LIN {X 0,Y 382.984,Z 108.401,A -85,B 0,C 180,E1 -11921.35,E2 -11921.35} C_VEL
LIN {X 0,Y 382.996,Z 108.402,A -85,B 0,C 180,E1 -11924.306,E2 -11924.306} C_VEL
LIN {X 0,Y 383.012,Z 108.398,A -85,B 0,C 180,E1 -11927.243,E2 -11927.243} C_VEL
LIN {X 0,Y 383.015,Z 108.397,A -85,B 0,C 180,E1 -11930.417,E2 -11930.417} C_VEL
LIN {X 0,Y 383.027,Z 108.398,A -85,B 0,C 180,E1 -11934.047,E2 -11934.047} C_VEL
LIN {X 0,Y 382.99,Z 108.406,A -85,B 0,C 180,E1 -11937.581,E2 -11937.581} C_VEL
LIN {X 0,Y 383.007,Z 108.425,A -85,B 0,C 180,E1 -11939.047,E2 -11939.047} C_VEL
LIN {X 0,Y 386.008,Z 121.95,A -85,B 0,C 180,E1 -11942.044,E2 -11942.044} C_VEL
LIN {X 0,Y 387.468,Z 129.298,A -85,B 0,C 180,E1 -11943.618,E2 -11943.618} C_VEL
LIN {X 0,Y 387.156,Z 135.337,A -85,B 0,C 180,E1 -11944.808,E2 -11944.808} C_VEL
LIN {X 0,Y 386.879,Z 138.646,A -85,B 0,C 180,E1 -11945.451,E2 -11945.451} C_VEL
LIN {X 0,Y 392.631,Z 173.743,A -85,B 0,C 180,E1 -11946.461,E2 -11946.461} C_VEL
LIN {X 0,Y 390.831,Z 276.351,A -85,B 0,C 180,E1 -11948.37,E2 -11948.37} C_VEL
LIN {X 0,Y 390.139,Z 291.161,A -85,B 0,C 180,E1 -11948.85,E2 -11948.85} C_VEL
LIN {X 0,Y 389.232,Z 305.249,A -85,B 0,C 180,E1 -11949.524,E2 -11949.524} C_VEL
LIN {X 0,Y 388.275,Z 318.604,A -85,B 0,C 180,E1 -11950.388,E2 -11950.388} C_VEL
LIN {X 0,Y 387.128,Z 331.76,A -85,B 0,C 180,E1 -11951.478,E2 -11951.478} C_VEL
LIN {X 0,Y 386.001,Z 343.198,A -85,B 0,C 180,E1 -11952.656,E2 -11952.656} C_VEL
LIN {X 0,Y 384.821,Z 354.677,A -85,B 0,C 180,E1 -11954.102,E2 -11954.102} C_VEL
LIN {X 0,Y 383.88,Z 365.216,A -85,B 0,C 180,E1 -11955.747,E2 -11955.747} C_VEL
LIN {X 0,Y 383.141,Z 373.396,A -85,B 0,C 180,E1 -11957.286,E2 -11957.286} C_VEL
LIN {X 0,Y 382.412,Z 381.481,A -85,B 0,C 180,E1 -11959.144,E2 -11959.144} C_VEL
LIN {X 0,Y 381.982,Z 387.982,A -85,B 0,C 180,E1 -11961.004,E2 -11961.004} C_VEL
LIN {X 0,Y 381.708,Z 393.729,A -85,B 0,C 180,E1 -11963.128,E2 -11963.128} C_VEL
LIN {X 0,Y 381.584,Z 396.98,A -85,B 0,C 180,E1 -11964.718,E2 -11964.718} C_VEL
LIN {X 0,Y 381.596,Z 398.675,A -85,B 0,C 180,E1 -11965.777,E2 -11965.777} C_VEL
LIN {X 0,Y 381.561,Z 401.002,A -85,B 0,C 180,E1 -11967.89,E2 -11967.89} C_VEL
LIN {X 0,Y 381.643,Z 401.969,A -85,B 0,C 180,E1 -11970.002,E2 -11970.002} C_VEL
LIN {X 0,Y 381.557,Z 401.592,A -85,B 0,C 180,E1 -11972.113,E2 -11972.113} C_VEL
LIN {X 0,Y 381.601,Z 399.883,A -85,B 0,C 180,E1 -11974.226,E2 -11974.226} C_VEL
LIN {X 0,Y 381.711,Z 396.809,A -85,B 0,C 180,E1 -11976.344,E2 -11976.344} C_VEL
LIN {X 0,Y 381.981,Z 392.289,A -85,B 0,C 180,E1 -11978.466,E2 -11978.466} C_VEL
LIN {X 0,Y 382.349,Z 387.826,A -85,B 0,C 180,E1 -11980.058,E2 -11980.058} C_VEL
LIN {X 0,Y 383.09,Z 381.408,A -85,B 0,C 180,E1 -11981.912,E2 -11981.912} C_VEL
LIN {X 0,Y 383.97,Z 373.46,A -85,B 0,C 180,E1 -11983.767,E2 -11983.767} C_VEL
LIN {X 0,Y 384.983,Z 365.183,A -85,B 0,C 180,E1 -11985.351,E2 -11985.351} C_VEL
LIN {X 0,Y 386.295,Z 355.246,A -85,B 0,C 180,E1 -11986.925,E2 -11986.925} C_VEL
LIN {X 0,Y 387.796,Z 344.222,A -85,B 0,C 180,E1 -11988.355,E2 -11988.355} C_VEL
LIN {X 0,Y 389.296,Z 331.93,A -85,B 0,C 180,E1 -11989.649,E2 -11989.649} C_VEL
LIN {X 0,Y 390.757,Z 318.639,A -85,B 0,C 180,E1 -11990.761,E2 -11990.761} C_VEL
LIN {X 0,Y 392.043,Z 305.232,A -85,B 0,C 180,E1 -11991.632,E2 -11991.632} C_VEL
LIN {X 0,Y 393.105,Z 291.561,A -85,B 0,C 180,E1 -11992.295,E2 -11992.295} C_VEL
LIN {X 0,Y 393.962,Z 277.474,A -85,B 0,C 180,E1 -11992.763,E2 -11992.763} C_VEL
LIN {X 0,Y 394.874,Z 240.379,A -85,B 0,C 180,E1 -11993.487,E2 -11993.487} C_VEL
LIN {X 0,Y 396.111,Z 173.208,A -85,B 0,C 180,E1 -11994.759,E2 -11994.759} C_VEL
LIN {X 0,Y 392.055,Z 152.238,A -85,B 0,C 180,E1 -11995.513,E2 -11995.513} C_VEL
LIN {X 0,Y 388.852,Z 138.136,A -85,B 0,C 180,E1 -11996.083,E2 -11996.083} C_VEL
LIN {X 0,Y 389.136,Z 134.462,A -85,B 0,C 180,E1 -11996.842,E2 -11996.842} C_VEL
LIN {X 0,Y 386.935,Z 123.671,A -85,B 0,C 180,E1 -11999.369,E2 -11999.369} C_VEL
LIN {X 0,Y 383.951,Z 111.962,A -85,B 0,C 180,E1 -12002.306,E2 -12002.306} C_VEL
LIN {X 0,Y 383.025,Z 108.405,A -85,B 0,C 180,E1 -12003.274,E2 -12003.274} C_VEL
LIN {X 0,Y 383.037,Z 108.402,A -85,B 0,C 180,E1 -12006.162,E2 -12006.162} C_VEL
LIN {X 0,Y 383.002,Z 108.395,A -85,B 0,C 180,E1 -12009.961,E2 -12009.961} C_VEL
LIN {X 0,Y 383.021,Z 108.398,A -85,B 0,C 180,E1 -12012.778,E2 -12012.778} C_VEL
LIN {X 0,Y 383.011,Z 108.401,A -85,B 0,C 180,E1 -12015.788,E2 -12015.788} C_VEL
LIN {X 0,Y 382.986,Z 108.385,A -85,B 0,C 180,E1 -12018.798,E2 -12018.798} C_VEL
LIN {X 0,Y 383.009,Z 108.397,A -85,B 0,C 180,E1 -12022.096,E2 -12022.096} C_VEL
LIN {X 0,Y 383.026,Z 108.396,A -85,B 0,C 180,E1 -12025.33,E2 -12025.33} C_VEL
LIN {X 0,Y 382.996,Z 108.398,A -85,B 0,C 180,E1 -12029.08,E2 -12029.08} C_VEL
LIN {X 0,Y 383.007,Z 108.394,A -85,B 0,C 180,E1 -12032.691,E2 -12032.691} C_VEL
LIN {X 0,Y 383.031,Z 108.389,A -85,B 0,C 180,E1 -12036.19,E2 -12036.19} C_VEL
LIN {X 0,Y 383.069,Z 108.384,A -85,B 0,C 180,E1 -12039.596,E2 -12039.596} C_VEL
LIN {X 0,Y 383.118,Z 108.384,A -85,B 0,C 180,E1 -12042.929,E2 -12042.929} C_VEL
LIN {X 0,Y 383.138,Z 108.387,A -85,B 0,C 180,E1 -12046.461,E2 -12046.461} C_VEL
LIN {X 0,Y 383.154,Z 108.386,A -85,B 0,C 180,E1 -12050.495,E2 -12050.495} C_VEL
LIN {X 0,Y 383.252,Z 108.366,A -85,B 0,C 180,E1 -12053.68,E2 -12053.68} C_VEL
LIN {X 0,Y 383.388,Z 108.348,A -85,B 0,C 180,E1 -12057.896,E2 -12057.896} C_VEL
LIN {X 0,Y 383.521,Z 108.336,A -85,B 0,C 180,E1 -12059.997,E2 -12059.997} C_VEL
LIN {X 0,Y 383.244,Z 108.37,A -85,B 0,C 180,E1 -12063.15,E2 -12063.15} C_VEL
LIN {X 0,Y 383.244,Z 108.369,A -85,B 0,C 180,E1 -12066.489,E2 -12066.489} C_VEL
LIN {X 0,Y 383.147,Z 108.378,A -85,B 0,C 180,E1 -12069.498,E2 -12069.498} C_VEL
LIN {X 0,Y 383.138,Z 108.38,A -85,B 0,C 180,E1 -12072.712,E2 -12072.712} C_VEL
LIN {X 0,Y 383.08,Z 108.388,A -85,B 0,C 180,E1 -12075.969,E2 -12075.969} C_VEL
LIN {X 0,Y 383.058,Z 108.394,A -85,B 0,C 180,E1 -12079.279,E2 -12079.279} C_VEL
LIN {X 0,Y 382.991,Z 108.402,A -85,B 0,C 180,E1 -12082.661,E2 -12082.661} C_VEL
LIN {X 0,Y 383.073,Z 108.387,A -85,B 0,C 180,E1 -12086.119,E2 -12086.119} C_VEL
LIN {X 0,Y 382.98,Z 108.387,A -85,B 0,C 180,E1 -12089.696,E2 -12089.696} C_VEL
LIN {X 0,Y 382.992,Z 108.395,A -85,B 0,C 180,E1 -12093.396,E2 -12093.396} C_VEL
LIN {X 0,Y 383.019,Z 108.402,A -85,B 0,C 180,E1 -12096.16,E2 -12096.16} C_VEL
LIN {X 0,Y 382.993,Z 108.404,A -85,B 0,C 180,E1 -12099.954,E2 -12099.954} C_VEL
LIN {X 0,Y 382.989,Z 108.404,A -85,B 0,C 180,E1 -12102.774,E2 -12102.774} C_VEL
LIN {X 0,Y 383,Z 108.566,A -85,B 0,C 180,E1 -12104.476,E2 -12104.476} C_VEL
LIN {X 0,Y 385.879,Z 120.269,A -85,B 0,C 180,E1 -12107.716,E2 -12107.716} C_VEL
LIN {X 0,Y 394.419,Z 139.311,A -85,B 0,C 180,E1 -12108.835,E2 -12108.835} C_VEL
LIN {X 0,Y 396.68,Z 148.471,A -85,B 0,C 180,E1 -12109.205,E2 -12109.205} C_VEL
LIN {X 0,Y 394.376,Z 256.219,A -85,B 0,C 180,E1 -12111.247,E2 -12111.247} C_VEL
LIN {X 0,Y 393.662,Z 270.685,A -85,B 0,C 180,E1 -12111.716,E2 -12111.716} C_VEL
LIN {X 0,Y 392.707,Z 284.97,A -85,B 0,C 180,E1 -12112.407,E2 -12112.407} C_VEL
LIN {X 0,Y 391.631,Z 297.377,A -85,B 0,C 180,E1 -12113.205,E2 -12113.205} C_VEL
LIN {X 0,Y 390.409,Z 309.653,A -85,B 0,C 180,E1 -12114.21,E2 -12114.21} C_VEL
LIN {X 0,Y 388.934,Z 321.956,A -85,B 0,C 180,E1 -12115.461,E2 -12115.461} C_VEL
LIN {X 0,Y 387.528,Z 333.02,A -85,B 0,C 180,E1 -12116.85,E2 -12116.85} C_VEL
LIN {X 0,Y 386.183,Z 342.972,A -85,B 0,C 180,E1 -12118.372,E2 -12118.372} C_VEL
LIN {X 0,Y 384.838,Z 352.497,A -85,B 0,C 180,E1 -12120.154,E2 -12120.154} C_VEL
LIN {X 0,Y 383.855,Z 359.942,A -85,B 0,C 180,E1 -12121.87,E2 -12121.87} C_VEL
LIN {X 0,Y 382.976,Z 366.892,A -85,B 0,C 180,E1 -12123.868,E2 -12123.868} C_VEL
LIN {X 0,Y 382.423,Z 371.625,A -85,B 0,C 180,E1 -12125.574,E2 -12125.574} C_VEL
LIN {X 0,Y 382.064,Z 375.285,A -85,B 0,C 180,E1 -12127.275,E2 -12127.275} C_VEL
LIN {X 0,Y 381.84,Z 377.212,A -85,B 0,C 180,E1 -12128.399,E2 -12128.399} C_VEL
LIN {X 0,Y 381.64,Z 379.115,A -85,B 0,C 180,E1 -12129.898,E2 -12129.898} C_VEL
LIN {X 0,Y 381.451,Z 380.58,A -85,B 0,C 180,E1 -12131.746,E2 -12131.746} C_VEL
LIN {X 0,Y 381.415,Z 380.992,A -85,B 0,C 180,E1 -12133.954,E2 -12133.954} C_VEL
LIN {X 0,Y 381.43,Z 379.994,A -85,B 0,C 180,E1 -12136.14,E2 -12136.14} C_VEL
LIN {X 0,Y 381.541,Z 378.714,A -85,B 0,C 180,E1 -12137.466,E2 -12137.466} C_VEL
LIN {X 0,Y 381.699,Z 375.859,A -85,B 0,C 180,E1 -12139.388,E2 -12139.388} C_VEL
LIN {X 0,Y 382.025,Z 371.264,A -85,B 0,C 180,E1 -12141.535,E2 -12141.535} C_VEL
LIN {X 0,Y 382.379,Z 366.428,A -85,B 0,C 180,E1 -12143.232,E2 -12143.232} C_VEL
LIN {X 0,Y 382.979,Z 359.141,A -85,B 0,C 180,E1 -12145.262,E2 -12145.262} C_VEL
LIN {X 0,Y 383.816,Z 350.737,A -85,B 0,C 180,E1 -12147.112,E2 -12147.112} C_VEL
LIN {X 0,Y 384.69,Z 341.997,A -85,B 0,C 180,E1 -12148.69,E2 -12148.69} C_VEL
LIN {X 0,Y 385.77,Z 331.417,A -85,B 0,C 180,E1 -12150.259,E2 -12150.259} C_VEL
LIN {X 0,Y 386.927,Z 319.878,A -85,B 0,C 180,E1 -12151.656,E2 -12151.656} C_VEL
LIN {X 0,Y 387.903,Z 309.107,A -85,B 0,C 180,E1 -12152.724,E2 -12152.724} C_VEL
LIN {X 0,Y 388.937,Z 296.319,A -85,B 0,C 180,E1 -12153.754,E2 -12153.754} C_VEL
LIN {X 0,Y 389.601,Z 286.012,A -85,B 0,C 180,E1 -12154.42,E2 -12154.42} C_VEL
LIN {X 0,Y 389.359,Z 280.539,A -85,B 0,C 180,E1 -12154.748,E2 -12154.748} C_VEL
LIN {X 0,Y 387.044,Z 271.618,A -85,B 0,C 180,E1 -12155.294,E2 -12155.294} C_VEL
LIN {X 0,Y 384.646,Z 262.541,A -85,B 0,C 180,E1 -12155.769,E2 -12155.769} C_VEL
LIN {X 0,Y 384.14,Z 256.824,A -85,B 0,C 180,E1 -12155.969,E2 -12155.969} C_VEL
LIN {X 0,Y 386.292,Z 148.656,A -85,B 0,C 180,E1 -12158.013,E2 -12158.013} C_VEL
LIN {X 0,Y 383.004,Z 132.931,A -85,B 0,C 180,E1 -12158.511,E2 -12158.511} C_VEL
LIN {X 0,Y 378.282,Z 119.77,A -85,B 0,C 180,E1 -12159.075,E2 -12159.075} C_VEL
LIN {X 0,Y 376.073,Z 109.269,A -85,B 0,C 180,E1 -12161.724,E2 -12161.724} C_VEL
LIN {X 0,Y 376.043,Z 109.266,A -85,B 0,C 180,E1 -12165.166,E2 -12165.166} C_VEL
LIN {X 0,Y 376.001,Z 109.27,A -85,B 0,C 180,E1 -12168.525,E2 -12168.525} C_VEL
LIN {X 0,Y 375.988,Z 109.274,A -85,B 0,C 180,E1 -12171.951,E2 -12171.951} C_VEL
LIN {X 0,Y 375.972,Z 109.279,A -85,B 0,C 180,E1 -12175.462,E2 -12175.462} C_VEL
LIN {X 0,Y 375.942,Z 109.282,A -85,B 0,C 180,E1 -12179.08,E2 -12179.08} C_VEL
LIN {X 0,Y 375.924,Z 109.283,A -85,B 0,C 180,E1 -12182.829,E2 -12182.829} C_VEL
LIN {X 0,Y 375.985,Z 109.274,A -85,B 0,C 180,E1 -12186.517,E2 -12186.517} C_VEL
LIN {X 0,Y 375.983,Z 109.272,A -85,B 0,C 180,E1 -12189.978,E2 -12189.978} C_VEL
LIN {X 0,Y 375.977,Z 109.273,A -85,B 0,C 180,E1 -12193.757,E2 -12193.757} C_VEL
LIN {X 0,Y 375.974,Z 109.279,A -85,B 0,C 180,E1 -12196.802,E2 -12196.802} C_VEL
LIN {X 0,Y 375.971,Z 109.275,A -85,B 0,C 180,E1 -12200.03,E2 -12200.03} C_VEL
LIN {X 0,Y 375.938,Z 109.278,A -85,B 0,C 180,E1 -12203.498,E2 -12203.498} C_VEL
LIN {X 0,Y 375.934,Z 109.28,A -85,B 0,C 180,E1 -12205.892,E2 -12205.892} C_VEL
LIN {X 0,Y 375.951,Z 109.277,A -85,B 0,C 180,E1 -12209.691,E2 -12209.691} C_VEL
LIN {X 0,Y 375.98,Z 109.279,A -85,B 0,C 180,E1 -12212.145,E2 -12212.145} C_VEL
LIN {X 0,Y 375.987,Z 109.274,A -85,B 0,C 180,E1 -12214.542,E2 -12214.542} C_VEL
LIN {X 0,Y 376.005,Z 109.276,A -85,B 0,C 180,E1 -12218.053,E2 -12218.053} C_VEL
LIN {X 0,Y 376.014,Z 109.271,A -85,B 0,C 180,E1 -12221.478,E2 -12221.478} C_VEL
LIN {X 0,Y 376.045,Z 109.265,A -85,B 0,C 180,E1 -12224.836,E2 -12224.836} C_VEL
LIN {X 0,Y 376.043,Z 109.267,A -85,B 0,C 180,E1 -12228.14,E2 -12228.14} C_VEL
LIN {X 0,Y 376.243,Z 109.244,A -85,B 0,C 180,E1 -12231.881,E2 -12231.881} C_VEL
LIN {X 0,Y 376.162,Z 109.25,A -85,B 0,C 180,E1 -12234.643,E2 -12234.643} C_VEL
LIN {X 0,Y 376.343,Z 109.23,A -85,B 0,C 180,E1 -12237.863,E2 -12237.863} C_VEL
LIN {X 0,Y 376.48,Z 109.211,A -85,B 0,C 180,E1 -12240.004,E2 -12240.004} C_VEL
LIN {X 0,Y 376.181,Z 109.254,A -85,B 0,C 180,E1 -12243.216,E2 -12243.216} C_VEL
LIN {X 0,Y 376.238,Z 109.241,A -85,B 0,C 180,E1 -12246.438,E2 -12246.438} C_VEL
LIN {X 0,Y 376.197,Z 109.247,A -85,B 0,C 180,E1 -12248.599,E2 -12248.599} C_VEL
LIN {X 0,Y 376.043,Z 109.265,A -85,B 0,C 180,E1 -12251.867,E2 -12251.867} C_VEL
LIN {X 0,Y 376.052,Z 109.267,A -85,B 0,C 180,E1 -12255.171,E2 -12255.171} C_VEL
LIN {X 0,Y 376.019,Z 109.272,A -85,B 0,C 180,E1 -12258.529,E2 -12258.529} C_VEL
LIN {X 0,Y 375.959,Z 109.276,A -85,B 0,C 180,E1 -12261.957,E2 -12261.957} C_VEL
LIN {X 0,Y 376.003,Z 109.27,A -85,B 0,C 180,E1 -12265.464,E2 -12265.464} C_VEL
LIN {X 0,Y 375.968,Z 109.275,A -85,B 0,C 180,E1 -12269.082,E2 -12269.082} C_VEL
LIN {X 0,Y 375.948,Z 109.278,A -85,B 0,C 180,E1 -12272.832,E2 -12272.832} C_VEL
LIN {X 0,Y 375.956,Z 109.276,A -85,B 0,C 180,E1 -12275.418,E2 -12275.418} C_VEL
LIN {X 0,Y 375.973,Z 109.279,A -85,B 0,C 180,E1 -12278.273,E2 -12278.273} C_VEL
LIN {X 0,Y 375.934,Z 109.28,A -85,B 0,C 180,E1 -12281.603,E2 -12281.603} C_VEL
LIN {X 0,Y 375.928,Z 109.28,A -85,B 0,C 180,E1 -12285.271,E2 -12285.271} C_VEL
LIN {X 0,Y 375.936,Z 109.28,A -85,B 0,C 180,E1 -12288.402,E2 -12288.402} C_VEL
LIN {X 0,Y 375.974,Z 109.28,A -85,B 0,C 180,E1 -12291.733,E2 -12291.733} C_VEL
LIN {X 0,Y 375.983,Z 109.276,A -85,B 0,C 180,E1 -12295.335,E2 -12295.335} C_VEL
LIN {X 0,Y 375.98,Z 109.303,A -85,B 0,C 180,E1 -12298.724,E2 -12298.724} C_VEL
LIN {X 0,Y 378.954,Z 122.797,A -85,B 0,C 180,E1 -12301.778,E2 -12301.778} C_VEL
LIN {X 0,Y 380.608,Z 131.627,A -85,B 0,C 180,E1 -12303.696,E2 -12303.696} C_VEL
LIN {X 0,Y 380.067,Z 138.479,A -85,B 0,C 180,E1 -12305.06,E2 -12305.06} C_VEL
LIN {X 0,Y 385.957,Z 174.406,A -85,B 0,C 180,E1 -12306.114,E2 -12306.114} C_VEL
LIN {X 0,Y 384.092,Z 276.228,A -85,B 0,C 180,E1 -12308.042,E2 -12308.042} C_VEL
LIN {X 0,Y 383.433,Z 290.253,A -85,B 0,C 180,E1 -12308.497,E2 -12308.497} C_VEL
LIN {X 0,Y 382.544,Z 303.967,A -85,B 0,C 180,E1 -12309.15,E2 -12309.15} C_VEL
LIN {X 0,Y 381.528,Z 317.567,A -85,B 0,C 180,E1 -12310.027,E2 -12310.027} C_VEL
LIN {X 0,Y 380.349,Z 330.897,A -85,B 0,C 180,E1 -12311.135,E2 -12311.135} C_VEL
LIN {X 0,Y 379.032,Z 343.647,A -85,B 0,C 180,E1 -12312.466,E2 -12312.466} C_VEL
LIN {X 0,Y 377.937,Z 354.056,A -85,B 0,C 180,E1 -12313.805,E2 -12313.805} C_VEL
LIN {X 0,Y 376.95,Z 364.385,A -85,B 0,C 180,E1 -12315.424,E2 -12315.424} C_VEL
LIN {X 0,Y 376.181,Z 372.926,A -85,B 0,C 180,E1 -12317.046,E2 -12317.046} C_VEL
LIN {X 0,Y 375.391,Z 381.06,A -85,B 0,C 180,E1 -12318.938,E2 -12318.938} C_VEL
LIN {X 0,Y 374.917,Z 387.606,A -85,B 0,C 180,E1 -12320.833,E2 -12320.833} C_VEL
LIN {X 0,Y 374.638,Z 393.396,A -85,B 0,C 180,E1 -12322.998,E2 -12322.998} C_VEL
LIN {X 0,Y 374.494,Z 396.686,A -85,B 0,C 180,E1 -12324.617,E2 -12324.617} C_VEL
LIN {X 0,Y 374.451,Z 399.753,A -85,B 0,C 180,E1 -12326.774,E2 -12326.774} C_VEL
LIN {X 0,Y 374.52,Z 401.432,A -85,B 0,C 180,E1 -12328.926,E2 -12328.926} C_VEL
LIN {X 0,Y 374.558,Z 401.764,A -85,B 0,C 180,E1 -12330.002,E2 -12330.002} C_VEL
LIN {X 0,Y 374.455,Z 401.421,A -85,B 0,C 180,E1 -12332.153,E2 -12332.153} C_VEL
LIN {X 0,Y 374.505,Z 399.746,A -85,B 0,C 180,E1 -12334.306,E2 -12334.306} C_VEL
LIN {X 0,Y 374.632,Z 396.707,A -85,B 0,C 180,E1 -12336.464,E2 -12336.464} C_VEL
LIN {X 0,Y 374.936,Z 392.225,A -85,B 0,C 180,E1 -12338.626,E2 -12338.626} C_VEL
LIN {X 0,Y 375.323,Z 387.807,A -85,B 0,C 180,E1 -12340.248,E2 -12340.248} C_VEL
LIN {X 0,Y 376.119,Z 381.442,A -85,B 0,C 180,E1 -12342.136,E2 -12342.136} C_VEL
LIN {X 0,Y 377.059,Z 373.556,A -85,B 0,C 180,E1 -12344.024,E2 -12344.024} C_VEL
LIN {X 0,Y 378.129,Z 365.341,A -85,B 0,C 180,E1 -12345.636,E2 -12345.636} C_VEL
LIN {X 0,Y 379.499,Z 355.475,A -85,B 0,C 180,E1 -12347.237,E2 -12347.237} C_VEL
LIN {X 0,Y 381.084,Z 344.535,A -85,B 0,C 180,E1 -12348.69,E2 -12348.69} C_VEL
LIN {X 0,Y 382.646,Z 332.407,A -85,B 0,C 180,E1 -12350.005,E2 -12350.005} C_VEL
LIN {X 0,Y 384.155,Z 319.32,A -85,B 0,C 180,E1 -12351.132,E2 -12351.132} C_VEL
LIN {X 0,Y 385.497,Z 306.109,A -85,B 0,C 180,E1 -12352.018,E2 -12352.018} C_VEL
LIN {X 0,Y 386.595,Z 292.812,A -85,B 0,C 180,E1 -12352.691,E2 -12352.691} C_VEL
LIN {X 0,Y 387.539,Z 278.34,A -85,B 0,C 180,E1 -12353.197,E2 -12353.197} C_VEL
LIN {X 0,Y 388.129,Z 256.717,A -85,B 0,C 180,E1 -12353.654,E2 -12353.654} C_VEL
LIN {X 0,Y 389.863,Z 174.36,A -85,B 0,C 180,E1 -12355.23,E2 -12355.23} C_VEL
LIN {X 0,Y 385.895,Z 153.716,A -85,B 0,C 180,E1 -12355.992,E2 -12355.992} C_VEL
LIN {X 0,Y 382.313,Z 137.821,A -85,B 0,C 180,E1 -12356.671,E2 -12356.671} C_VEL
LIN {X 0,Y 382.077,Z 134.655,A -85,B 0,C 180,E1 -12357.379,E2 -12357.379} C_VEL
LIN {X 0,Y 379.758,Z 123.915,A -85,B 0,C 180,E1 -12359.98,E2 -12359.98} C_VEL
LIN {X 0,Y 376.83,Z 112.5,A -85,B 0,C 180,E1 -12362.934,E2 -12362.934} C_VEL
LIN {X 0,Y 375.995,Z 109.279,A -85,B 0,C 180,E1 -12363.827,E2 -12363.827} C_VEL
LIN {X 0,Y 375.963,Z 109.276,A -85,B 0,C 180,E1 -12366.742,E2 -12366.742} C_VEL
LIN {X 0,Y 375.984,Z 109.269,A -85,B 0,C 180,E1 -12369.967,E2 -12369.967} C_VEL
LIN {X 0,Y 375.944,Z 109.281,A -85,B 0,C 180,E1 -12373.766,E2 -12373.766} C_VEL
LIN {X 0,Y 375.949,Z 109.28,A -85,B 0,C 180,E1 -12376.81,E2 -12376.81} C_VEL
LIN {X 0,Y 375.956,Z 109.277,A -85,B 0,C 180,E1 -12380.534,E2 -12380.534} C_VEL
LIN {X 0,Y 375.973,Z 109.275,A -85,B 0,C 180,E1 -12383.496,E2 -12383.496} C_VEL
LIN {X 0,Y 375.972,Z 109.273,A -85,B 0,C 180,E1 -12385.887,E2 -12385.887} C_VEL
LIN {X 0,Y 375.977,Z 109.276,A -85,B 0,C 180,E1 -12389.686,E2 -12389.686} C_VEL
LIN {X 0,Y 375.948,Z 109.279,A -85,B 0,C 180,E1 -12393.34,E2 -12393.34} C_VEL
LIN {X 0,Y 375.992,Z 109.27,A -85,B 0,C 180,E1 -12396.885,E2 -12396.885} C_VEL
LIN {X 0,Y 376.01,Z 109.264,A -85,B 0,C 180,E1 -12400.337,E2 -12400.337} C_VEL
LIN {X 0,Y 376.041,Z 109.26,A -85,B 0,C 180,E1 -12403.716,E2 -12403.716} C_VEL
LIN {X 0,Y 376.116,Z 109.256,A -85,B 0,C 180,E1 -12407.039,E2 -12407.039} C_VEL
LIN {X 0,Y 376.124,Z 109.259,A -85,B 0,C 180,E1 -12410.315,E2 -12410.315} C_VEL
LIN {X 0,Y 376.21,Z 109.243,A -85,B 0,C 180,E1 -12413.561,E2 -12413.561} C_VEL
LIN {X 0,Y 376.353,Z 109.224,A -85,B 0,C 180,E1 -12417.856,E2 -12417.856} C_VEL
LIN {X 0,Y 376.491,Z 109.211,A -85,B 0,C 180,E1 -12419.996,E2 -12419.996} C_VEL
LIN {X 0,Y 376.356,Z 109.225,A -85,B 0,C 180,E1 -12422.137,E2 -12422.137} C_VEL
LIN {X 0,Y 376.214,Z 109.246,A -85,B 0,C 180,E1 -12426.473,E2 -12426.473} C_VEL
LIN {X 0,Y 376.117,Z 109.254,A -85,B 0,C 180,E1 -12429.678,E2 -12429.678} C_VEL
LIN {X 0,Y 376.091,Z 109.258,A -85,B 0,C 180,E1 -12433.653,E2 -12433.653} C_VEL
LIN {X 0,Y 376.042,Z 109.267,A -85,B 0,C 180,E1 -12437.602,E2 -12437.602} C_VEL
LIN {X 0,Y 375.976,Z 109.272,A -85,B 0,C 180,E1 -12440.828,E2 -12440.828} C_VEL
LIN {X 0,Y 375.982,Z 109.275,A -85,B 0,C 180,E1 -12444.277,E2 -12444.277} C_VEL
LIN {X 0,Y 376.013,Z 109.268,A -85,B 0,C 180,E1 -12446.648,E2 -12446.648} C_VEL
LIN {X 0,Y 375.955,Z 109.263,A -85,B 0,C 180,E1 -12450.308,E2 -12450.308} C_VEL
LIN {X 0,Y 375.949,Z 109.268,A -85,B 0,C 180,E1 -12454.107,E2 -12454.107} C_VEL
LIN {X 0,Y 375.94,Z 109.28,A -85,B 0,C 180,E1 -12456.737,E2 -12456.737} C_VEL
LIN {X 0,Y 375.973,Z 109.278,A -85,B 0,C 180,E1 -12459.966,E2 -12459.966} C_VEL
LIN {X 0,Y 375.932,Z 109.366,A -85,B 0,C 180,E1 -12463.912,E2 -12463.912} C_VEL
LIN {X 0,Y 378.716,Z 120.544,A -85,B 0,C 180,E1 -12467.083,E2 -12467.083} C_VEL
LIN {X 0,Y 386.709,Z 137.791,A -85,B 0,C 180,E1 -12468.163,E2 -12468.163} C_VEL
LIN {X 0,Y 389.117,Z 143.905,A -85,B 0,C 180,E1 -12468.495,E2 -12468.495} C_VEL
LIN {X 0,Y 390.521,Z 150.476,A -85,B 0,C 180,E1 -12468.749,E2 -12468.749} C_VEL
LIN {X 0,Y 388.016,Z 257.036,A -85,B 0,C 180,E1 -12470.799,E2 -12470.799} C_VEL
LIN {X 0,Y 387.315,Z 270.742,A -85,B 0,C 180,E1 -12471.253,E2 -12471.253} C_VEL
LIN {X 0,Y 386.422,Z 283.832,A -85,B 0,C 180,E1 -12471.884,E2 -12471.884} C_VEL
LIN {X 0,Y 385.337,Z 296.147,A -85,B 0,C 180,E1 -12472.666,E2 -12472.666} C_VEL
LIN {X 0,Y 383.991,Z 309.047,A -85,B 0,C 180,E1 -12473.717,E2 -12473.717} C_VEL
LIN {X 0,Y 382.436,Z 321.185,A -85,B 0,C 180,E1 -12474.949,E2 -12474.949} C_VEL
LIN {X 0,Y 380.913,Z 332.633,A -85,B 0,C 180,E1 -12476.39,E2 -12476.39} C_VEL
LIN {X 0,Y 379.576,Z 341.992,A -85,B 0,C 180,E1 -12477.821,E2 -12477.821} C_VEL
LIN {X 0,Y 378.188,Z 351.452,A -85,B 0,C 180,E1 -12479.574,E2 -12479.574} C_VEL
LIN {X 0,Y 377.049,Z 359.405,A -85,B 0,C 180,E1 -12481.388,E2 -12481.388} C_VEL
LIN {X 0,Y 376.145,Z 366.327,A -85,B 0,C 180,E1 -12483.356,E2 -12483.356} C_VEL
LIN {X 0,Y 375.473,Z 371.175,A -85,B 0,C 180,E1 -12485.091,E2 -12485.091} C_VEL
LIN {X 0,Y 375.086,Z 374.98,A -85,B 0,C 180,E1 -12486.827,E2 -12486.827} C_VEL
LIN {X 0,Y 374.647,Z 378.597,A -85,B 0,C 180,E1 -12489.118,E2 -12489.118} C_VEL
LIN {X 0,Y 374.377,Z 380.662,A -85,B 0,C 180,E1 -12491.388,E2 -12491.388} C_VEL
LIN {X 0,Y 374.344,Z 381.228,A -85,B 0,C 180,E1 -12493.642,E2 -12493.642} C_VEL
LIN {X 0,Y 374.327,Z 380.377,A -85,B 0,C 180,E1 -12495.871,E2 -12495.871} C_VEL
LIN {X 0,Y 374.488,Z 378.121,A -85,B 0,C 180,E1 -12498.085,E2 -12498.085} C_VEL
LIN {X 0,Y 374.74,Z 374.435,A -85,B 0,C 180,E1 -12500.281,E2 -12500.281} C_VEL
LIN {X 0,Y 375.119,Z 369.231,A -85,B 0,C 180,E1 -12502.463,E2 -12502.463} C_VEL
LIN {X 0,Y 375.506,Z 364.187,A -85,B 0,C 180,E1 -12504.09,E2 -12504.09} C_VEL
LIN {X 0,Y 376.165,Z 356.982,A -85,B 0,C 180,E1 -12505.981,E2 -12505.981} C_VEL
LIN {X 0,Y 377.013,Z 349.425,A -85,B 0,C 180,E1 -12507.595,E2 -12507.595} C_VEL
LIN {X 0,Y 377.959,Z 340.377,A -85,B 0,C 180,E1 -12509.199,E2 -12509.199} C_VEL
LIN {X 0,Y 379.099,Z 329.436,A -85,B 0,C 180,E1 -12510.795,E2 -12510.795} C_VEL
LIN {X 0,Y 380.215,Z 318.307,A -85,B 0,C 180,E1 -12512.117,E2 -12512.117} C_VEL
LIN {X 0,Y 381.337,Z 306.025,A -85,B 0,C 180,E1 -12513.3,E2 -12513.3} C_VEL
LIN {X 0,Y 382.292,Z 294.241,A -85,B 0,C 180,E1 -12514.216,E2 -12514.216} C_VEL
LIN {X 0,Y 383.167,Z 281.411,A -85,B 0,C 180,E1 -12514.997,E2 -12514.997} C_VEL
LIN {X 0,Y 383.801,Z 267.802,A -85,B 0,C 180,E1 -12515.614,E2 -12515.614} C_VEL
LIN {X 0,Y 384.14,Z 256.824,A -85,B 0,C 180,E1 -12515.969,E2 -12515.969} C_VEL
LIN {X 0,Y 383.696,Z 251.057,A -85,B 0,C 180,E1 -12516.149,E2 -12516.149} C_VEL
LIN {X 0,Y 378.665,Z 232.321,A -85,B 0,C 180,E1 -12516.775,E2 -12516.775} C_VEL
LIN {X 0,Y 378.102,Z 226.503,A -85,B 0,C 180,E1 -12516.915,E2 -12516.915} C_VEL
LIN {X 0,Y 379.542,Z 148.9,A -85,B 0,C 180,E1 -12518.391,E2 -12518.391} C_VEL
LIN {X 0,Y 376.586,Z 135.147,A -85,B 0,C 180,E1 -12518.843,E2 -12518.843} C_VEL
LIN {X 0,Y 371.124,Z 120.022,A -85,B 0,C 180,E1 -12519.499,E2 -12519.499} C_VEL
LIN {X 0,Y 369.014,Z 110.148,A -85,B 0,C 180,E1 -12522.022,E2 -12522.022} C_VEL
LIN {X 0,Y 368.996,Z 110.144,A -85,B 0,C 180,E1 -12524.334,E2 -12524.334} C_VEL
LIN {X 0,Y 369,Z 110.147,A -85,B 0,C 180,E1 -12527.785,E2 -12527.785} C_VEL
LIN {X 0,Y 368.951,Z 110.152,A -85,B 0,C 180,E1 -12531.217,E2 -12531.217} C_VEL
LIN {X 0,Y 368.926,Z 110.153,A -85,B 0,C 180,E1 -12534.776,E2 -12534.776} C_VEL
LIN {X 0,Y 368.951,Z 110.149,A -85,B 0,C 180,E1 -12538.436,E2 -12538.436} C_VEL
LIN {X 0,Y 368.876,Z 110.158,A -85,B 0,C 180,E1 -12542.238,E2 -12542.238} C_VEL
LIN {X 0,Y 368.905,Z 110.16,A -85,B 0,C 180,E1 -12545.005,E2 -12545.005} C_VEL
LIN {X 0,Y 368.953,Z 110.151,A -85,B 0,C 180,E1 -12548.657,E2 -12548.657} C_VEL
LIN {X 0,Y 368.912,Z 110.154,A -85,B 0,C 180,E1 -12552.022,E2 -12552.022} C_VEL
LIN {X 0,Y 368.971,Z 110.148,A -85,B 0,C 180,E1 -12555.197,E2 -12555.197} C_VEL
LIN {X 0,Y 368.912,Z 110.155,A -85,B 0,C 180,E1 -12558.188,E2 -12558.188} C_VEL
LIN {X 0,Y 368.885,Z 110.157,A -85,B 0,C 180,E1 -12561.361,E2 -12561.361} C_VEL
LIN {X 0,Y 368.91,Z 110.154,A -85,B 0,C 180,E1 -12565.149,E2 -12565.149} C_VEL
LIN {X 0,Y 368.904,Z 110.155,A -85,B 0,C 180,E1 -12569.05,E2 -12569.05} C_VEL
LIN {X 0,Y 368.964,Z 110.147,A -85,B 0,C 180,E1 -12571.568,E2 -12571.568} C_VEL
LIN {X 0,Y 368.941,Z 110.15,A -85,B 0,C 180,E1 -12575.228,E2 -12575.228} C_VEL
LIN {X 0,Y 368.97,Z 110.146,A -85,B 0,C 180,E1 -12578.955,E2 -12578.955} C_VEL
LIN {X 0,Y 368.975,Z 110.148,A -85,B 0,C 180,E1 -12582.261,E2 -12582.261} C_VEL
LIN {X 0,Y 369.02,Z 110.142,A -85,B 0,C 180,E1 -12586.231,E2 -12586.231} C_VEL
LIN {X 0,Y 369.057,Z 110.137,A -85,B 0,C 180,E1 -12590.135,E2 -12590.135} C_VEL
LIN {X 0,Y 369.174,Z 110.121,A -85,B 0,C 180,E1 -12592.346,E2 -12592.346} C_VEL
LIN {X 0,Y 369.134,Z 110.126,A -85,B 0,C 180,E1 -12594.541,E2 -12594.541} C_VEL
LIN {X 0,Y 369.308,Z 110.106,A -85,B 0,C 180,E1 -12597.822,E2 -12597.822} C_VEL
LIN {X 0,Y 369.449,Z 110.087,A -85,B 0,C 180,E1 -12600.004,E2 -12600.004} C_VEL
LIN {X 0,Y 369.309,Z 110.104,A -85,B 0,C 180,E1 -12602.185,E2 -12602.185} C_VEL
LIN {X 0,Y 369.2,Z 110.119,A -85,B 0,C 180,E1 -12606.562,E2 -12606.562} C_VEL
LIN {X 0,Y 369.13,Z 110.129,A -85,B 0,C 180,E1 -12608.764,E2 -12608.764} C_VEL
LIN {X 0,Y 368.998,Z 110.143,A -85,B 0,C 180,E1 -12612.097,E2 -12612.097} C_VEL
LIN {X 0,Y 368.992,Z 110.144,A -85,B 0,C 180,E1 -12615.468,E2 -12615.468} C_VEL
LIN {X 0,Y 368.977,Z 110.15,A -85,B 0,C 180,E1 -12618.896,E2 -12618.896} C_VEL
LIN {X 0,Y 368.929,Z 110.155,A -85,B 0,C 180,E1 -12622.398,E2 -12622.398} C_VEL
LIN {X 0,Y 368.997,Z 110.144,A -85,B 0,C 180,E1 -12625.983,E2 -12625.983} C_VEL
LIN {X 0,Y 368.959,Z 110.15,A -85,B 0,C 180,E1 -12628.815,E2 -12628.815} C_VEL
LIN {X 0,Y 368.896,Z 110.16,A -85,B 0,C 180,E1 -12632.241,E2 -12632.241} C_VEL
LIN {X 0,Y 368.928,Z 110.152,A -85,B 0,C 180,E1 -12635.004,E2 -12635.004} C_VEL
LIN {X 0,Y 368.908,Z 110.156,A -85,B 0,C 180,E1 -12638.643,E2 -12638.643} C_VEL
LIN {X 0,Y 368.882,Z 110.163,A -85,B 0,C 180,E1 -12642.012,E2 -12642.012} C_VEL
LIN {X 0,Y 368.881,Z 110.158,A -85,B 0,C 180,E1 -12645.178,E2 -12645.178} C_VEL
LIN {X 0,Y 368.884,Z 110.16,A -85,B 0,C 180,E1 -12648.18,E2 -12648.18} C_VEL
LIN {X 0,Y 368.908,Z 110.156,A -85,B 0,C 180,E1 -12651.363,E2 -12651.363} C_VEL
LIN {X 0,Y 368.939,Z 110.152,A -85,B 0,C 180,E1 -12655.149,E2 -12655.149} C_VEL
LIN {X 0,Y 368.956,Z 110.248,A -85,B 0,C 180,E1 -12658.407,E2 -12658.407} C_VEL
LIN {X 0,Y 372.235,Z 125.108,A -85,B 0,C 180,E1 -12661.837,E2 -12661.837} C_VEL
LIN {X 0,Y 373.629,Z 132.475,A -85,B 0,C 180,E1 -12663.467,E2 -12663.467} C_VEL
LIN {X 0,Y 373.263,Z 138.456,A -85,B 0,C 180,E1 -12664.662,E2 -12664.662} C_VEL
LIN {X 0,Y 379.287,Z 175.675,A -85,B 0,C 180,E1 -12665.77,E2 -12665.77} C_VEL
LIN {X 0,Y 377.383,Z 276.061,A -85,B 0,C 180,E1 -12667.703,E2 -12667.703} C_VEL
LIN {X 0,Y 376.701,Z 290.074,A -85,B 0,C 180,E1 -12668.165,E2 -12668.165} C_VEL
LIN {X 0,Y 375.791,Z 303.785,A -85,B 0,C 180,E1 -12668.829,E2 -12668.829} C_VEL
LIN {X 0,Y 374.753,Z 316.741,A -85,B 0,C 180,E1 -12669.671,E2 -12669.671} C_VEL
LIN {X 0,Y 373.564,Z 329.986,A -85,B 0,C 180,E1 -12670.779,E2 -12670.779} C_VEL
LIN {X 0,Y 372.31,Z 341.673,A -85,B 0,C 180,E1 -12671.996,E2 -12671.996} C_VEL
LIN {X 0,Y 371.266,Z 351.395,A -85,B 0,C 180,E1 -12673.223,E2 -12673.223} C_VEL
LIN {X 0,Y 370.152,Z 362.181,A -85,B 0,C 180,E1 -12674.868,E2 -12674.868} C_VEL
LIN {X 0,Y 369.348,Z 371.291,A -85,B 0,C 180,E1 -12676.566,E2 -12676.566} C_VEL
LIN {X 0,Y 368.507,Z 379.577,A -85,B 0,C 180,E1 -12678.45,E2 -12678.45} C_VEL
LIN {X 0,Y 367.986,Z 385.487,A -85,B 0,C 180,E1 -12680.104,E2 -12680.104} C_VEL
LIN {X 0,Y 367.7,Z 390.354,A -85,B 0,C 180,E1 -12681.76,E2 -12681.76} C_VEL
LIN {X 0,Y 367.486,Z 394.29,A -85,B 0,C 180,E1 -12683.413,E2 -12683.413} C_VEL
LIN {X 0,Y 367.406,Z 398.122,A -85,B 0,C 180,E1 -12685.613,E2 -12685.613} C_VEL
LIN {X 0,Y 367.361,Z 400.521,A -85,B 0,C 180,E1 -12687.809,E2 -12687.809} C_VEL
LIN {X 0,Y 367.461,Z 401.559,A -85,B 0,C 180,E1 -12690.002,E2 -12690.002} C_VEL
LIN {X 0,Y 367.356,Z 401.251,A -85,B 0,C 180,E1 -12692.194,E2 -12692.194} C_VEL
LIN {X 0,Y 367.414,Z 399.613,A -85,B 0,C 180,E1 -12694.39,E2 -12694.39} C_VEL
LIN {X 0,Y 367.562,Z 396.615,A -85,B 0,C 180,E1 -12696.589,E2 -12696.589} C_VEL
LIN {X 0,Y 367.869,Z 392.178,A -85,B 0,C 180,E1 -12698.793,E2 -12698.793} C_VEL
LIN {X 0,Y 368.445,Z 386.176,A -85,B 0,C 180,E1 -12700.998,E2 -12700.998} C_VEL
LIN {X 0,Y 369.432,Z 379.449,A -85,B 0,C 180,E1 -12702.918,E2 -12702.918} C_VEL
LIN {X 0,Y 370.461,Z 371.115,A -85,B 0,C 180,E1 -12704.84,E2 -12704.84} C_VEL
LIN {X 0,Y 371.709,Z 362.454,A -85,B 0,C 180,E1 -12706.477,E2 -12706.477} C_VEL
LIN {X 0,Y 373.264,Z 351.992,A -85,B 0,C 180,E1 -12708.101,E2 -12708.101} C_VEL
LIN {X 0,Y 374.997,Z 340.33,A -85,B 0,C 180,E1 -12709.574,E2 -12709.574} C_VEL
LIN {X 0,Y 376.578,Z 328.683,A -85,B 0,C 180,E1 -12710.77,E2 -12710.77} C_VEL
LIN {X 0,Y 378.048,Z 315.893,A -85,B 0,C 180,E1 -12711.828,E2 -12711.828} C_VEL
LIN {X 0,Y 379.418,Z 302.613,A -85,B 0,C 180,E1 -12712.677,E2 -12712.677} C_VEL
LIN {X 0,Y 380.541,Z 288.929,A -85,B 0,C 180,E1 -12713.325,E2 -12713.325} C_VEL
LIN {X 0,Y 381.408,Z 274.728,A -85,B 0,C 180,E1 -12713.772,E2 -12713.772} C_VEL
LIN {X 0,Y 383.657,Z 175.335,A -85,B 0,C 180,E1 -12715.721,E2 -12715.721} C_VEL
LIN {X 0,Y 379.01,Z 151.599,A -85,B 0,C 180,E1 -12716.633,E2 -12716.633} C_VEL
LIN {X 0,Y 375.624,Z 138.085,A -85,B 0,C 180,E1 -12717.238,E2 -12717.238} C_VEL
LIN {X 0,Y 375.368,Z 136.806,A -85,B 0,C 180,E1 -12717.476,E2 -12717.476} C_VEL
LIN {X 0,Y 373.212,Z 126.696,A -85,B 0,C 180,E1 -12719.973,E2 -12719.973} C_VEL
LIN {X 0,Y 370.276,Z 115.178,A -85,B 0,C 180,E1 -12723.01,E2 -12723.01} C_VEL
LIN {X 0,Y 368.955,Z 110.15,A -85,B 0,C 180,E1 -12724.439,E2 -12724.439} C_VEL
LIN {X 0,Y 368.912,Z 110.15,A -85,B 0,C 180,E1 -12727.564,E2 -12727.564} C_VEL
LIN {X 0,Y 368.921,Z 110.146,A -85,B 0,C 180,E1 -12730.37,E2 -12730.37} C_VEL
LIN {X 0,Y 368.897,Z 110.158,A -85,B 0,C 180,E1 -12733.615,E2 -12733.615} C_VEL
LIN {X 0,Y 368.901,Z 110.158,A -85,B 0,C 180,E1 -12736.695,E2 -12736.695} C_VEL
LIN {X 0,Y 368.922,Z 110.14,A -85,B 0,C 180,E1 -12739.643,E2 -12739.643} C_VEL
LIN {X 0,Y 368.911,Z 110.152,A -85,B 0,C 180,E1 -12743.144,E2 -12743.144} C_VEL
LIN {X 0,Y 368.91,Z 110.154,A -85,B 0,C 180,E1 -12746.46,E2 -12746.46} C_VEL
LIN {X 0,Y 368.928,Z 110.15,A -85,B 0,C 180,E1 -12749.043,E2 -12749.043} C_VEL
LIN {X 0,Y 368.931,Z 110.15,A -85,B 0,C 180,E1 -12751.557,E2 -12751.557} C_VEL
LIN {X 0,Y 368.947,Z 110.148,A -85,B 0,C 180,E1 -12755.221,E2 -12755.221} C_VEL
LIN {X 0,Y 368.934,Z 110.15,A -85,B 0,C 180,E1 -12758.978,E2 -12758.978} C_VEL
LIN {X 0,Y 369.004,Z 110.145,A -85,B 0,C 180,E1 -12762.255,E2 -12762.255} C_VEL
LIN {X 0,Y 369.05,Z 110.14,A -85,B 0,C 180,E1 -12766.225,E2 -12766.225} C_VEL
LIN {X 0,Y 369.074,Z 110.136,A -85,B 0,C 180,E1 -12770.129,E2 -12770.129} C_VEL
LIN {X 0,Y 369.171,Z 110.119,A -85,B 0,C 180,E1 -12773.438,E2 -12773.438} C_VEL
LIN {X 0,Y 369.317,Z 110.1,A -85,B 0,C 180,E1 -12777.815,E2 -12777.815} C_VEL
LIN {X 0,Y 369.461,Z 110.087,A -85,B 0,C 180,E1 -12779.996,E2 -12779.996} C_VEL
LIN {X 0,Y 369.321,Z 110.102,A -85,B 0,C 180,E1 -12782.177,E2 -12782.177} C_VEL
LIN {X 0,Y 369.178,Z 110.122,A -85,B 0,C 180,E1 -12786.555,E2 -12786.555} C_VEL
LIN {X 0,Y 369.067,Z 110.132,A -85,B 0,C 180,E1 -12789.864,E2 -12789.864} C_VEL
LIN {X 0,Y 369.039,Z 110.137,A -85,B 0,C 180,E1 -12793.768,E2 -12793.768} C_VEL
LIN {X 0,Y 369.001,Z 110.145,A -85,B 0,C 180,E1 -12797.764,E2 -12797.764} C_VEL
LIN {X 0,Y 368.926,Z 110.154,A -85,B 0,C 180,E1 -12801.215,E2 -12801.215} C_VEL
LIN {X 0,Y 368.948,Z 110.153,A -85,B 0,C 180,E1 -12804.771,E2 -12804.771} C_VEL
LIN {X 0,Y 368.956,Z 110.153,A -85,B 0,C 180,E1 -12807.199,E2 -12807.199} C_VEL
LIN {X 0,Y 368.902,Z 110.148,A -85,B 0,C 180,E1 -12810.983,E2 -12810.983} C_VEL
LIN {X 0,Y 368.925,Z 110.146,A -85,B 0,C 180,E1 -12814.849,E2 -12814.849} C_VEL
LIN {X 0,Y 368.893,Z 110.154,A -85,B 0,C 180,E1 -12818.635,E2 -12818.635} C_VEL
LIN {X 0,Y 368.866,Z 110.163,A -85,B 0,C 180,E1 -12822.005,E2 -12822.005} C_VEL
LIN {X 0,Y 368.904,Z 110.282,A -85,B 0,C 180,E1 -12823.35,E2 -12823.35} C_VEL
LIN {X 0,Y 371.533,Z 120.715,A -85,B 0,C 180,E1 -12826.405,E2 -12826.405} C_VEL
LIN {X 0,Y 380.044,Z 138.63,A -85,B 0,C 180,E1 -12827.6,E2 -12827.6} C_VEL
LIN {X 0,Y 383.265,Z 146.562,A -85,B 0,C 180,E1 -12828.055,E2 -12828.055} C_VEL
LIN {X 0,Y 384.309,Z 151.154,A -85,B 0,C 180,E1 -12828.243,E2 -12828.243} C_VEL
LIN {X 0,Y 381.698,Z 257.424,A -85,B 0,C 180,E1 -12830.321,E2 -12830.321} C_VEL
LIN {X 0,Y 380.939,Z 271.545,A -85,B 0,C 180,E1 -12830.803,E2 -12830.803} C_VEL
LIN {X 0,Y 379.972,Z 284.731,A -85,B 0,C 180,E1 -12831.456,E2 -12831.456} C_VEL
LIN {X 0,Y 378.863,Z 296.902,A -85,B 0,C 180,E1 -12832.253,E2 -12832.253} C_VEL
LIN {X 0,Y 377.611,Z 307.945,A -85,B 0,C 180,E1 -12833.151,E2 -12833.151} C_VEL
LIN {X 0,Y 375.995,Z 320.458,A -85,B 0,C 180,E1 -12834.423,E2 -12834.423} C_VEL
LIN {X 0,Y 374.413,Z 332.056,A -85,B 0,C 180,E1 -12835.889,E2 -12835.889} C_VEL
LIN {X 0,Y 373.074,Z 340.737,A -85,B 0,C 180,E1 -12837.206,E2 -12837.206} C_VEL
LIN {X 0,Y 371.592,Z 350.375,A -85,B 0,C 180,E1 -12838.975,E2 -12838.975} C_VEL
LIN {X 0,Y 370.31,Z 358.483,A -85,B 0,C 180,E1 -12840.8,E2 -12840.8} C_VEL
LIN {X 0,Y 369.316,Z 365.687,A -85,B 0,C 180,E1 -12842.823,E2 -12842.823} C_VEL
LIN {X 0,Y 368.567,Z 370.71,A -85,B 0,C 180,E1 -12844.592,E2 -12844.592} C_VEL
LIN {X 0,Y 368.088,Z 374.765,A -85,B 0,C 180,E1 -12846.403,E2 -12846.403} C_VEL
LIN {X 0,Y 367.612,Z 378.463,A -85,B 0,C 180,E1 -12848.699,E2 -12848.699} C_VEL
LIN {X 0,Y 367.479,Z 379.762,A -85,B 0,C 180,E1 -12849.863,E2 -12849.863} C_VEL
LIN {X 0,Y 367.243,Z 381.245,A -85,B 0,C 180,E1 -12852.168,E2 -12852.168} C_VEL
LIN {X 0,Y 367.261,Z 381.443,A -85,B 0,C 180,E1 -12853.317,E2 -12853.317} C_VEL
LIN {X 0,Y 367.213,Z 380.758,A -85,B 0,C 180,E1 -12855.592,E2 -12855.592} C_VEL
LIN {X 0,Y 367.375,Z 378.646,A -85,B 0,C 180,E1 -12857.851,E2 -12857.851} C_VEL
LIN {X 0,Y 367.61,Z 375.109,A -85,B 0,C 180,E1 -12860.091,E2 -12860.091} C_VEL
LIN {X 0,Y 367.991,Z 370.059,A -85,B 0,C 180,E1 -12862.316,E2 -12862.316} C_VEL
LIN {X 0,Y 368.405,Z 365.177,A -85,B 0,C 180,E1 -12863.976,E2 -12863.976} C_VEL
LIN {X 0,Y 369.057,Z 358.151,A -85,B 0,C 180,E1 -12865.903,E2 -12865.903} C_VEL
LIN {X 0,Y 370.043,Z 349.445,A -85,B 0,C 180,E1 -12867.822,E2 -12867.822} C_VEL
LIN {X 0,Y 371.026,Z 340.362,A -85,B 0,C 180,E1 -12869.456,E2 -12869.456} C_VEL
LIN {X 0,Y 372.232,Z 329.369,A -85,B 0,C 180,E1 -12871.08,E2 -12871.08} C_VEL
LIN {X 0,Y 373.37,Z 318.179,A -85,B 0,C 180,E1 -12872.426,E2 -12872.426} C_VEL
LIN {X 0,Y 374.435,Z 307.349,A -85,B 0,C 180,E1 -12873.496,E2 -12873.496} C_VEL
LIN {X 0,Y 375.397,Z 295.811,A -85,B 0,C 180,E1 -12874.428,E2 -12874.428} C_VEL
LIN {X 0,Y 376.366,Z 282.224,A -85,B 0,C 180,E1 -12875.289,E2 -12875.289} C_VEL
LIN {X 0,Y 377.009,Z 268.882,A -85,B 0,C 180,E1 -12875.917,E2 -12875.917} C_VEL
LIN {X 0,Y 377.468,Z 255.584,A -85,B 0,C 180,E1 -12876.345,E2 -12876.345} C_VEL
LIN {X 0,Y 378.102,Z 226.503,A -85,B 0,C 180,E1 -12876.915,E2 -12876.915} C_VEL
LIN {X 0,Y 377.543,Z 220.695,A -85,B 0,C 180,E1 -12877.061,E2 -12877.061} C_VEL
LIN {X 0,Y 372.525,Z 201.988,A -85,B 0,C 180,E1 -12877.718,E2 -12877.718} C_VEL
LIN {X 0,Y 372.05,Z 196.179,A -85,B 0,C 180,E1 -12877.864,E2 -12877.864} C_VEL
LIN {X 0,Y 372.848,Z 149.496,A -85,B 0,C 180,E1 -12878.773,E2 -12878.773} C_VEL
LIN {X 0,Y 370.298,Z 137.675,A -85,B 0,C 180,E1 -12879.172,E2 -12879.172} C_VEL
LIN {X 0,Y 363.921,Z 120.18,A -85,B 0,C 180,E1 -12879.952,E2 -12879.952} C_VEL
LIN {X 0,Y 361.959,Z 111.029,A -85,B 0,C 180,E1 -12882.331,E2 -12882.331} C_VEL
LIN {X 0,Y 361.962,Z 111.019,A -85,B 0,C 180,E1 -12884.619,E2 -12884.619} C_VEL
LIN {X 0,Y 361.938,Z 111.024,A -85,B 0,C 180,E1 -12888.099,E2 -12888.099} C_VEL
LIN {X 0,Y 361.896,Z 111.032,A -85,B 0,C 180,E1 -12891.651,E2 -12891.651} C_VEL
LIN {X 0,Y 361.895,Z 111.033,A -85,B 0,C 180,E1 -12895.291,E2 -12895.291} C_VEL
LIN {X 0,Y 361.887,Z 111.03,A -85,B 0,C 180,E1 -12897.779,E2 -12897.779} C_VEL
LIN {X 0,Y 361.826,Z 111.038,A -85,B 0,C 180,E1 -12901.628,E2 -12901.628} C_VEL
LIN {X 0,Y 361.853,Z 111.036,A -85,B 0,C 180,E1 -12905.349,E2 -12905.349} C_VEL
LIN {X 0,Y 361.904,Z 111.028,A -85,B 0,C 180,E1 -12908.418,E2 -12908.418} C_VEL
LIN {X 0,Y 361.874,Z 111.032,A -85,B 0,C 180,E1 -12911.322,E2 -12911.322} C_VEL
LIN {X 0,Y 361.909,Z 111.028,A -85,B 0,C 180,E1 -12914.352,E2 -12914.352} C_VEL
LIN {X 0,Y 361.858,Z 111.032,A -85,B 0,C 180,E1 -12917.561,E2 -12917.561} C_VEL
LIN {X 0,Y 361.847,Z 111.036,A -85,B 0,C 180,E1 -12920.975,E2 -12920.975} C_VEL
LIN {X 0,Y 361.848,Z 111.037,A -85,B 0,C 180,E1 -12924.658,E2 -12924.658} C_VEL
LIN {X 0,Y 361.836,Z 111.041,A -85,B 0,C 180,E1 -12928.376,E2 -12928.376} C_VEL
LIN {X 0,Y 361.9,Z 111.033,A -85,B 0,C 180,E1 -12932.225,E2 -12932.225} C_VEL
LIN {X 0,Y 361.911,Z 111.029,A -85,B 0,C 180,E1 -12935.876,E2 -12935.876} C_VEL
LIN {X 0,Y 361.91,Z 111.028,A -85,B 0,C 180,E1 -12939.545,E2 -12939.545} C_VEL
LIN {X 0,Y 361.917,Z 111.025,A -85,B 0,C 180,E1 -12943.07,E2 -12943.07} C_VEL
LIN {X 0,Y 361.983,Z 111.017,A -85,B 0,C 180,E1 -12946.531,E2 -12946.531} C_VEL
LIN {X 0,Y 362.021,Z 111.015,A -85,B 0,C 180,E1 -12949.942,E2 -12949.942} C_VEL
LIN {X 0,Y 362.137,Z 110.998,A -85,B 0,C 180,E1 -12952.196,E2 -12952.196} C_VEL
LIN {X 0,Y 362.107,Z 111.001,A -85,B 0,C 180,E1 -12954.435,E2 -12954.435} C_VEL
LIN {X 0,Y 362.272,Z 110.983,A -85,B 0,C 180,E1 -12957.78,E2 -12957.78} C_VEL
LIN {X 0,Y 362.419,Z 110.963,A -85,B 0,C 180,E1 -12960.004,E2 -12960.004} C_VEL
LIN {X 0,Y 362.273,Z 110.98,A -85,B 0,C 180,E1 -12962.227,E2 -12962.227} C_VEL
LIN {X 0,Y 362.164,Z 110.996,A -85,B 0,C 180,E1 -12966.69,E2 -12966.69} C_VEL
LIN {X 0,Y 362.066,Z 111.011,A -85,B 0,C 180,E1 -12968.937,E2 -12968.937} C_VEL
LIN {X 0,Y 361.953,Z 111.021,A -85,B 0,C 180,E1 -12972.336,E2 -12972.336} C_VEL
LIN {X 0,Y 361.956,Z 111.023,A -85,B 0,C 180,E1 -12974.624,E2 -12974.624} C_VEL
LIN {X 0,Y 361.955,Z 111.021,A -85,B 0,C 180,E1 -12978.103,E2 -12978.103} C_VEL
LIN {X 0,Y 361.888,Z 111.028,A -85,B 0,C 180,E1 -12981.656,E2 -12981.656} C_VEL
LIN {X 0,Y 361.925,Z 111.024,A -85,B 0,C 180,E1 -12985.293,E2 -12985.293} C_VEL
LIN {X 0,Y 361.916,Z 111.025,A -85,B 0,C 180,E1 -12987.781,E2 -12987.781} C_VEL
LIN {X 0,Y 361.845,Z 111.034,A -85,B 0,C 180,E1 -12991.288,E2 -12991.288} C_VEL
LIN {X 0,Y 361.853,Z 111.039,A -85,B 0,C 180,E1 -12994.284,E2 -12994.284} C_VEL
LIN {X 0,Y 361.863,Z 111.031,A -85,B 0,C 180,E1 -12997.226,E2 -12997.226} C_VEL
LIN {X 0,Y 361.835,Z 111.036,A -85,B 0,C 180,E1 -13000.758,E2 -13000.758} C_VEL
LIN {X 0,Y 361.818,Z 111.039,A -85,B 0,C 180,E1 -13004.371,E2 -13004.371} C_VEL
LIN {X 0,Y 361.838,Z 111.038,A -85,B 0,C 180,E1 -13007.571,E2 -13007.571} C_VEL
LIN {X 0,Y 361.869,Z 111.031,A -85,B 0,C 180,E1 -13010.977,E2 -13010.977} C_VEL
LIN {X 0,Y 361.877,Z 111.03,A -85,B 0,C 180,E1 -13014.658,E2 -13014.658} C_VEL
LIN {X 0,Y 361.896,Z 111.06,A -85,B 0,C 180,E1 -13018.051,E2 -13018.051} C_VEL
LIN {X 0,Y 365.114,Z 125.674,A -85,B 0,C 180,E1 -13021.494,E2 -13021.494} C_VEL
LIN {X 0,Y 366.622,Z 133.318,A -85,B 0,C 180,E1 -13023.227,E2 -13023.227} C_VEL
LIN {X 0,Y 366.421,Z 138.087,A -85,B 0,C 180,E1 -13024.226,E2 -13024.226} C_VEL
LIN {X 0,Y 372.581,Z 175.229,A -85,B 0,C 180,E1 -13025.376,E2 -13025.376} C_VEL
LIN {X 0,Y 370.685,Z 275.893,A -85,B 0,C 180,E1 -13027.351,E2 -13027.351} C_VEL
LIN {X 0,Y 369.914,Z 290.657,A -85,B 0,C 180,E1 -13027.853,E2 -13027.853} C_VEL
LIN {X 0,Y 368.925,Z 304.735,A -85,B 0,C 180,E1 -13028.562,E2 -13028.562} C_VEL
LIN {X 0,Y 367.82,Z 318.466,A -85,B 0,C 180,E1 -13029.5,E2 -13029.5} C_VEL
LIN {X 0,Y 366.646,Z 330.516,A -85,B 0,C 180,E1 -13030.548,E2 -13030.548} C_VEL
LIN {X 0,Y 365.362,Z 342.076,A -85,B 0,C 180,E1 -13031.787,E2 -13031.787} C_VEL
LIN {X 0,Y 364.164,Z 352.685,A -85,B 0,C 180,E1 -13033.175,E2 -13033.175} C_VEL
LIN {X 0,Y 363.069,Z 363.228,A -85,B 0,C 180,E1 -13034.853,E2 -13034.853} C_VEL
LIN {X 0,Y 362.269,Z 371.914,A -85,B 0,C 180,E1 -13036.54,E2 -13036.54} C_VEL
LIN {X 0,Y 361.387,Z 380.181,A -85,B 0,C 180,E1 -13038.504,E2 -13038.504} C_VEL
LIN {X 0,Y 360.809,Z 386.828,A -85,B 0,C 180,E1 -13040.472,E2 -13040.472} C_VEL
LIN {X 0,Y 360.538,Z 391.423,A -85,B 0,C 180,E1 -13042.159,E2 -13042.159} C_VEL
LIN {X 0,Y 360.332,Z 396.085,A -85,B 0,C 180,E1 -13044.405,E2 -13044.405} C_VEL
LIN {X 0,Y 360.286,Z 399.231,A -85,B 0,C 180,E1 -13046.647,E2 -13046.647} C_VEL
LIN {X 0,Y 360.32,Z 400.983,A -85,B 0,C 180,E1 -13048.884,E2 -13048.884} C_VEL
LIN {X 0,Y 360.364,Z 401.353,A -85,B 0,C 180,E1 -13050.002,E2 -13050.002} C_VEL
LIN {X 0,Y 360.261,Z 401.083,A -85,B 0,C 180,E1 -13052.238,E2 -13052.238} C_VEL
LIN {X 0,Y 360.326,Z 399.484,A -85,B 0,C 180,E1 -13054.476,E2 -13054.476} C_VEL
LIN {X 0,Y 360.493,Z 396.525,A -85,B 0,C 180,E1 -13056.719,E2 -13056.719} C_VEL
LIN {X 0,Y 360.818,Z 392.13,A -85,B 0,C 180,E1 -13058.966,E2 -13058.966} C_VEL
LIN {X 0,Y 361.434,Z 386.181,A -85,B 0,C 180,E1 -13061.214,E2 -13061.214} C_VEL
LIN {X 0,Y 362.484,Z 379.509,A -85,B 0,C 180,E1 -13063.17,E2 -13063.17} C_VEL
LIN {X 0,Y 363.577,Z 371.255,A -85,B 0,C 180,E1 -13065.128,E2 -13065.128} C_VEL
LIN {X 0,Y 364.901,Z 362.675,A -85,B 0,C 180,E1 -13066.794,E2 -13066.794} C_VEL
LIN {X 0,Y 366.527,Z 352.311,A -85,B 0,C 180,E1 -13068.446,E2 -13068.446} C_VEL
LIN {X 0,Y 368.336,Z 340.752,A -85,B 0,C 180,E1 -13069.943,E2 -13069.943} C_VEL
LIN {X 0,Y 370.129,Z 327.964,A -85,B 0,C 180,E1 -13071.281,E2 -13071.281} C_VEL
LIN {X 0,Y 371.737,Z 314.872,A -85,B 0,C 180,E1 -13072.365,E2 -13072.365} C_VEL
LIN {X 0,Y 373.116,Z 301.329,A -85,B 0,C 180,E1 -13073.229,E2 -13073.229} C_VEL
LIN {X 0,Y 374.355,Z 287.073,A -85,B 0,C 180,E1 -13073.88,E2 -13073.88} C_VEL
LIN {X 0,Y 375.181,Z 273.243,A -85,B 0,C 180,E1 -13074.302,E2 -13074.302} C_VEL
LIN {X 0,Y 377.502,Z 176.962,A -85,B 0,C 180,E1 -13076.212,E2 -13076.212} C_VEL
LIN {X 0,Y 373.785,Z 157.285,A -85,B 0,C 180,E1 -13076.98,E2 -13076.98} C_VEL
LIN {X 0,Y 370.13,Z 141.774,A -85,B 0,C 180,E1 -13077.67,E2 -13077.67} C_VEL
LIN {X 0,Y 368.312,Z 137.329,A -85,B 0,C 180,E1 -13077.98,E2 -13077.98} C_VEL
LIN {X 0,Y 366.338,Z 128.159,A -85,B 0,C 180,E1 -13080.307,E2 -13080.307} C_VEL
LIN {X 0,Y 363.167,Z 115.744,A -85,B 0,C 180,E1 -13083.678,E2 -13083.678} C_VEL
LIN {X 0,Y 361.888,Z 111.03,A -85,B 0,C 180,E1 -13085.051,E2 -13085.051} C_VEL
LIN {X 0,Y 361.86,Z 111.035,A -85,B 0,C 180,E1 -13088.428,E2 -13088.428} C_VEL
LIN {X 0,Y 361.835,Z 111.033,A -85,B 0,C 180,E1 -13091.331,E2 -13091.331} C_VEL
LIN {X 0,Y 361.832,Z 111.04,A -85,B 0,C 180,E1 -13094.368,E2 -13094.368} C_VEL
LIN {X 0,Y 361.847,Z 111.027,A -85,B 0,C 180,E1 -13097.568,E2 -13097.568} C_VEL
LIN {X 0,Y 361.845,Z 111.036,A -85,B 0,C 180,E1 -13100.98,E2 -13100.98} C_VEL
LIN {X 0,Y 361.885,Z 111.031,A -85,B 0,C 180,E1 -13104.655,E2 -13104.655} C_VEL
LIN {X 0,Y 361.852,Z 111.032,A -85,B 0,C 180,E1 -13108.369,E2 -13108.369} C_VEL
LIN {X 0,Y 361.881,Z 111.034,A -85,B 0,C 180,E1 -13110.95,E2 -13110.95} C_VEL
LIN {X 0,Y 361.905,Z 111.031,A -85,B 0,C 180,E1 -13114.705,E2 -13114.705} C_VEL
LIN {X 0,Y 361.875,Z 111.033,A -85,B 0,C 180,E1 -13118.343,E2 -13118.343} C_VEL
LIN {X 0,Y 361.981,Z 111.019,A -85,B 0,C 180,E1 -13122.059,E2 -13122.059} C_VEL
LIN {X 0,Y 362.011,Z 111.016,A -85,B 0,C 180,E1 -13126.099,E2 -13126.099} C_VEL
LIN {X 0,Y 362.011,Z 111.014,A -85,B 0,C 180,E1 -13129.934,E2 -13129.934} C_VEL
LIN {X 0,Y 362.134,Z 110.996,A -85,B 0,C 180,E1 -13133.31,E2 -13133.31} C_VEL
LIN {X 0,Y 362.28,Z 110.976,A -85,B 0,C 180,E1 -13137.773,E2 -13137.773} C_VEL
LIN {X 0,Y 362.409,Z 110.965,A -85,B 0,C 180,E1 -13139.996,E2 -13139.996} C_VEL
LIN {X 0,Y 362.284,Z 110.979,A -85,B 0,C 180,E1 -13142.22,E2 -13142.22} C_VEL
LIN {X 0,Y 362.14,Z 110.999,A -85,B 0,C 180,E1 -13146.683,E2 -13146.683} C_VEL
LIN {X 0,Y 362.003,Z 111.013,A -85,B 0,C 180,E1 -13150.059,E2 -13150.059} C_VEL
LIN {X 0,Y 362,Z 111.014,A -85,B 0,C 180,E1 -13153.894,E2 -13153.894} C_VEL
LIN {X 0,Y 361.967,Z 111.023,A -85,B 0,C 180,E1 -13157.934,E2 -13157.934} C_VEL
LIN {X 0,Y 361.887,Z 111.033,A -85,B 0,C 180,E1 -13161.648,E2 -13161.648} C_VEL
LIN {X 0,Y 361.921,Z 111.026,A -85,B 0,C 180,E1 -13165.286,E2 -13165.286} C_VEL
LIN {X 0,Y 361.901,Z 111.029,A -85,B 0,C 180,E1 -13167.774,E2 -13167.774} C_VEL
LIN {X 0,Y 361.829,Z 111.04,A -85,B 0,C 180,E1 -13171.625,E2 -13171.625} C_VEL
LIN {X 0,Y 361.863,Z 111.031,A -85,B 0,C 180,E1 -13175.34,E2 -13175.34} C_VEL
LIN {X 0,Y 361.854,Z 111.036,A -85,B 0,C 180,E1 -13179.022,E2 -13179.022} C_VEL
LIN {X 0,Y 361.839,Z 111.2,A -85,B 0,C 180,E1 -13182.754,E2 -13182.754} C_VEL
LIN {X 0,Y 364.344,Z 120.992,A -85,B 0,C 180,E1 -13185.707,E2 -13185.707} C_VEL
LIN {X 0,Y 373.312,Z 139.408,A -85,B 0,C 180,E1 -13187.001,E2 -13187.001} C_VEL
LIN {X 0,Y 377.4,Z 149.233,A -85,B 0,C 180,E1 -13187.595,E2 -13187.595} C_VEL
LIN {X 0,Y 378.147,Z 152.91,A -85,B 0,C 180,E1 -13187.743,E2 -13187.743} C_VEL
LIN {X 0,Y 375.424,Z 257.512,A -85,B 0,C 180,E1 -13189.818,E2 -13189.818} C_VEL
LIN {X 0,Y 374.668,Z 271.205,A -85,B 0,C 180,E1 -13190.286,E2 -13190.286} C_VEL
LIN {X 0,Y 373.668,Z 284.422,A -85,B 0,C 180,E1 -13190.943,E2 -13190.943} C_VEL
LIN {X 0,Y 372.391,Z 297.651,A -85,B 0,C 180,E1 -13191.823,E2 -13191.823} C_VEL
LIN {X 0,Y 370.976,Z 309.606,A -85,B 0,C 180,E1 -13192.834,E2 -13192.834} C_VEL
LIN {X 0,Y 369.41,Z 321.017,A -85,B 0,C 180,E1 -13194.026,E2 -13194.026} C_VEL
LIN {X 0,Y 367.755,Z 332.437,A -85,B 0,C 180,E1 -13195.498,E2 -13195.498} C_VEL
LIN {X 0,Y 366.34,Z 341.181,A -85,B 0,C 180,E1 -13196.854,E2 -13196.854} C_VEL
LIN {X 0,Y 364.768,Z 350.765,A -85,B 0,C 180,E1 -13198.652,E2 -13198.652} C_VEL
LIN {X 0,Y 363.458,Z 358.647,A -85,B 0,C 180,E1 -13200.464,E2 -13200.464} C_VEL
LIN {X 0,Y 362.487,Z 365.039,A -85,B 0,C 180,E1 -13202.268,E2 -13202.268} C_VEL
LIN {X 0,Y 361.708,Z 370.246,A -85,B 0,C 180,E1 -13204.075,E2 -13204.075} C_VEL
LIN {X 0,Y 361.057,Z 374.942,A -85,B 0,C 180,E1 -13206.172,E2 -13206.172} C_VEL
LIN {X 0,Y 360.601,Z 378.33,A -85,B 0,C 180,E1 -13208.264,E2 -13208.264} C_VEL
LIN {X 0,Y 360.273,Z 380.703,A -85,B 0,C 180,E1 -13210.631,E2 -13210.631} C_VEL
